C01832=1236.003,114.402,-48.327,-178.206,5.493,148.420
C01833=1235.998,114.651,-48.346,-178.204,5.494,148.419
C01834=1235.993,114.900,-48.366,-178.202,5.495,148.419
C01835=1235.989,115.150,-48.386,-178.199,5.496,148.418
C01836=1235.983,115.399,-48.405,-178.196,5.497,148.418
C01837=1235.979,115.648,-48.424,-178.194,5.498,148.417
C01838=1235.975,115.897,-48.444,-178.191,5.499,148.416
C01839=1235.969,116.146,-48.464,-178.189,5.500,148.416
C01840=1235.965,116.395,-48.483,-178.186,5.500,148.415
C01841=1235.960,116.645,-48.503,-178.183,5.502,148.415
C01842=1235.955,116.894,-48.522,-178.181,5.503,148.414
C01843=1235.950,117.143,-48.543,-178.178,5.503,148.414
C01844=1235.945,117.392,-48.562,-178.176,5.504,148.413
C01845=1235.940,117.641,-48.582,-178.174,5.505,148.413
C01846=1235.935,117.891,-48.601,-178.171,5.506,148.412
C01847=1235.932,118.139,-48.621,-178.168,5.507,148.412
C01848=1235.927,118.389,-48.641,-178.166,5.508,148.411
C01849=1235.921,118.638,-48.660,-178.163,5.509,148.410
C01850=1235.917,118.887,-48.680,-178.161,5.510,148.410
C01851=1235.912,119.136,-48.700,-178.158,5.511,148.409
C01852=1235.908,119.386,-48.720,-178.155,5.512,148.409
C01853=1235.903,119.634,-48.740,-178.153,5.513,148.408
C01854=1235.898,119.884,-48.759,-178.151,5.513,148.408
C01855=1235.893,120.133,-48.779,-178.148,5.514,148.407
C01856=1235.889,120.382,-48.799,-178.145,5.516,148.407
C01857=1235.883,120.631,-48.819,-178.143,5.517,148.406
C01858=1235.879,120.880,-48.838,-178.141,5.517,148.406
C01859=1235.874,121.129,-48.859,-178.138,5.518,148.405
C01860=1235.869,121.379,-48.878,-178.135,5.519,148.404
C01861=1235.864,121.627,-48.898,-178.133,5.521,148.404
C01862=1235.860,121.877,-48.918,-178.130,5.521,148.403
C01863=1235.855,122.126,-48.938,-178.128,5.522,148.403
C01864=1235.850,122.375,-48.958,-178.125,5.523,148.402
C01865=1235.845,122.624,-48.977,-178.122,5.524,148.402
C01866=1235.841,122.873,-48.998,-178.120,5.525,148.401
C01867=1235.836,123.123,-49.017,-178.117,5.526,148.401
C01868=1235.831,123.372,-49.038,-178.115,5.527,148.400
C01869=1235.827,123.621,-49.057,-178.113,5.528,148.399
C01870=1235.821,123.870,-49.078,-178.110,5.529,148.399
C01871=1235.816,124.119,-49.098,-178.107,5.530,148.398
C01872=1235.812,124.368,-49.118,-178.105,5.531,148.398
C01873=1235.807,124.618,-49.138,-178.102,5.531,148.397
C01874=1235.803,124.867,-49.158,-178.100,5.533,148.397
C01875=1235.798,125.116,-49.178,-178.097,5.534,148.396
C01876=1235.793,125.365,-49.198,-178.095,5.535,148.396
C01877=1235.788,125.614,-49.217,-178.092,5.535,148.395
C01878=1235.784,125.863,-49.238,-178.089,5.537,148.394
C01879=1235.779,126.113,-49.257,-178.087,5.538,148.394
C01880=1235.774,126.362,-49.278,-178.084,5.538,148.393
C01881=1235.769,126.611,-49.299,-178.082,5.539,148.393
C01882=1235.764,126.861,-49.318,-178.079,5.541,148.392
C01883=1235.759,127.109,-49.338,-178.076,5.542,148.392
C01884=1235.755,127.358,-49.358,-178.074,5.543,148.391
C01885=1235.750,127.607,-49.378,-178.072,5.543,148.391
C01886=1235.745,127.857,-49.399,-178.070,5.544,148.390
C01887=1235.740,128.106,-49.419,-178.066,5.546,148.390
C01888=1235.736,128.355,-49.439,-178.064,5.546,148.389
C01889=1235.731,128.604,-49.460,-178.062,5.547,148.389
C01890=1235.727,128.854,-49.480,-178.059,5.549,148.388
C01891=1235.722,129.102,-49.500,-178.056,5.550,148.388
C01892=1235.717,129.351,-49.520,-178.054,5.550,148.387
C01893=1235.712,129.601,-49.540,-178.052,5.551,148.387
C01894=1235.707,129.850,-49.561,-178.049,5.553,148.386
C01895=1235.703,130.099,-49.581,-178.046,5.553,148.385
C01896=1235.697,130.348,-49.601,-178.044,5.554,148.385
C01897=1235.693,130.597,-49.622,-178.041,5.555,148.384
C01898=1235.689,130.846,-49.642,-178.039,5.557,148.384
C01899=1235.684,131.095,-49.662,-178.036,5.558,148.383
C01900=1235.679,131.345,-49.683,-178.034,5.559,148.383
C01901=1235.674,131.594,-49.703,-178.031,5.559,148.382
C01902=1235.670,131.843,-49.723,-178.028,5.561,148.382
C01903=1235.665,132.091,-49.743,-178.026,5.562,148.381
C01904=1235.660,132.341,-49.764,-178.023,5.562,148.381
C01905=1235.655,132.590,-49.784,-178.021,5.564,148.380
C01906=1235.650,132.839,-49.804,-178.018,5.565,148.380
C01907=1235.645,133.088,-49.825,-178.016,5.566,148.379
C01908=1235.641,133.337,-49.846,-178.013,5.566,148.379
C01909=1235.635,133.606,-49.867,-178.010,5.568,148.378
C01910=1235.631,133.875,-49.889,-178.008,5.569,148.377
C01911=1235.626,134.143,-49.912,-178.005,5.570,148.377
C01912=1235.620,134.412,-49.934,-178.002,5.571,148.376
C01913=1235.616,134.661,-49.954,-177.999,5.572,148.376
C01914=1235.610,134.910,-49.975,-177.997,5.573,148.375
C01915=1235.606,135.159,-49.995,-177.995,5.574,148.375
C01916=1235.602,135.408,-50.016,-177.992,5.575,148.374
C01917=1235.596,135.658,-50.037,-177.989,5.577,148.374
C01918=1235.592,135.907,-50.057,-177.987,5.578,148.373
C01919=1235.588,136.156,-50.077,-177.985,5.578,148.373
C01920=1235.582,136.405,-50.098,-177.982,5.580,148.372
C01921=1235.578,136.654,-50.119,-177.979,5.581,148.372
C01922=1235.573,136.903,-50.140,-177.977,5.582,148.371
C01923=1235.568,137.152,-50.160,-177.974,5.583,148.371
C01924=1235.564,137.401,-50.180,-177.971,5.584,148.370
C01925=1235.559,137.650,-50.201,-177.969,5.585,148.370
C01926=1235.554,137.899,-50.222,-177.967,5.585,148.369
C01927=1235.549,138.148,-50.243,-177.964,5.587,148.369
C01928=1235.545,138.397,-50.263,-177.961,5.588,148.368
C01929=1235.539,138.647,-50.284,-177.959,5.589,148.368
C01930=1235.536,138.896,-50.305,-177.956,5.590,148.367
C01931=1235.530,139.145,-50.326,-177.954,5.591,148.367
C01932=1235.526,139.394,-50.346,-177.951,5.592,148.366
C01933=1235.521,139.644,-50.367,-177.949,5.594,148.366
C01934=1235.516,139.893,-50.387,-177.946,5.594,148.365
C01935=1235.512,140.142,-50.408,-177.944,5.595,148.364
C01936=1235.507,140.391,-50.429,-177.941,5.597,148.364
C01937=1235.502,140.640,-50.449,-177.939,5.598,148.363
C01938=1235.497,140.889,-50.470,-177.936,5.599,148.363
C01939=1235.493,141.138,-50.490,-177.934,5.600,148.362
C01940=1235.488,141.387,-50.512,-177.931,5.601,148.362
C01941=1235.483,141.636,-50.533,-177.929,5.602,148.361
C01942=1235.478,141.885,-50.553,-177.926,5.604,148.361
C01943=1235.474,142.135,-50.575,-177.923,5.604,148.360
C01944=1235.469,142.384,-50.595,-177.921,5.605,148.360
C01945=1235.464,142.633,-50.616,-177.918,5.607,148.359
C01946=1235.460,142.881,-50.637,-177.916,5.608,148.359
C01947=1235.455,143.131,-50.658,-177.913,5.608,148.358
C01948=1235.450,143.380,-50.679,-177.910,5.610,148.358
C01949=1235.445,143.629,-50.700,-177.908,5.611,148.357
C01950=1235.441,143.878,-50.720,-177.906,5.612,148.357
C01951=1235.436,144.127,-50.742,-177.903,5.613,148.356
C01952=1235.431,144.376,-50.763,-177.901,5.614,148.356
C01953=1235.427,144.625,-50.783,-177.898,5.615,148.355
C01954=1235.422,144.875,-50.804,-177.895,5.617,148.355
C01955=1235.418,145.123,-50.825,-177.893,5.617,148.354
C01956=1235.412,145.372,-50.846,-177.891,5.618,148.354
C01957=1235.407,145.621,-50.867,-177.887,5.620,148.353
C01958=1235.404,145.870,-50.889,-177.885,5.621,148.353
C01959=1235.399,146.120,-50.910,-177.883,5.622,148.352
C01960=1235.393,146.369,-50.931,-177.880,5.623,148.352
C01961=1235.389,146.617,-50.952,-177.878,5.624,148.351
C01962=1235.384,146.867,-50.973,-177.875,5.625,148.351
C01963=1235.379,147.116,-50.994,-177.873,5.627,148.350
C01964=1235.375,147.365,-51.015,-177.870,5.628,148.350
C01965=1235.370,147.614,-51.036,-177.867,5.629,148.349
C01966=1235.365,147.863,-51.057,-177.865,5.630,148.349
C01967=1235.361,148.112,-51.078,-177.863,5.631,148.348
C01968=1235.356,148.361,-51.099,-177.860,5.632,148.348
C01969=1235.351,148.610,-51.121,-177.857,5.633,148.347
C01970=1235.347,148.859,-51.142,-177.855,5.634,148.347
C01971=1235.342,149.109,-51.163,-177.852,5.636,148.346
C01972=1235.337,149.357,-51.184,-177.850,5.637,148.346
C01973=1235.332,149.607,-51.206,-177.847,5.638,148.345
C01974=1235.328,149.855,-51.227,-177.844,5.639,148.345
C01975=1235.323,150.105,-51.248,-177.842,5.640,148.344
C01976=1235.318,150.353,-51.269,-177.839,5.642,148.344
C01977=1235.313,150.603,-51.290,-177.837,5.643,148.343
C01978=1235.309,150.852,-51.312,-177.834,5.643,148.343
C01979=1235.304,151.101,-51.333,-177.832,5.645,148.342
C01980=1235.299,151.350,-51.354,-177.830,5.646,148.342
C01981=1235.294,151.599,-51.375,-177.826,5.648,148.341
C01982=1235.291,151.848,-51.397,-177.824,5.649,148.341
C01983=1235.286,152.097,-51.418,-177.822,5.649,148.340
C01984=1235.281,152.346,-51.439,-177.819,5.651,148.340
C01985=1235.276,152.596,-51.461,-177.817,5.652,148.339
C01986=1235.271,152.844,-51.482,-177.814,5.654,148.339
C01987=1235.266,153.093,-51.504,-177.811,5.654,148.338
C01988=1235.262,153.342,-51.524,-177.809,5.655,148.338
C01989=1235.258,153.591,-51.547,-177.806,5.657,148.337
C01990=1235.252,153.841,-51.568,-177.804,5.658,148.337
C01991=1235.248,154.089,-51.589,-177.801,5.660,148.337
C01992=1235.243,154.339,-51.611,-177.799,5.660,148.336
C01993=1235.238,154.588,-51.632,-177.797,5.661,148.336
C01994=1235.234,154.836,-51.653,-177.793,5.663,148.335
C01995=1235.229,155.085,-51.675,-177.791,5.664,148.335
C01996=1235.225,155.335,-51.696,-177.788,5.665,148.334
C01997=1235.220,155.583,-51.718,-177.786,5.666,148.334
C01998=1235.215,155.832,-51.740,-177.784,5.667,148.333
C01999=1235.210,156.082,-51.761,-177.781,5.669,148.333
C02000=1235.205,156.331,-51.783,-177.779,5.670,148.332
C02001=1235.201,156.579,-51.804,-177.776,5.671,148.332
C02002=1235.196,156.829,-51.826,-177.773,5.672,148.331
C02003=1235.191,157.078,-51.847,-177.770,5.674,148.331
C02004=1235.186,157.326,-51.869,-177.768,5.675,148.330
C02005=1235.183,157.575,-51.891,-177.766,5.676,148.330
C02006=1235.178,157.825,-51.911,-177.763,5.677,148.329
C02007=1235.173,158.073,-51.933,-177.761,5.678,148.329
C02008=1235.168,158.323,-51.955,-177.758,5.680,148.328
C02009=1235.164,158.571,-51.977,-177.756,5.681,148.328
C02010=1235.159,158.821,-51.999,-177.752,5.682,148.327
C02011=1235.154,159.070,-52.020,-177.750,5.683,148.327
C02012=1235.149,159.319,-52.042,-177.748,5.684,148.326
C02013=1235.144,159.587,-52.066,-177.745,5.686,148.326
C02014=1235.139,159.857,-52.089,-177.742,5.687,148.325
C02015=1235.134,160.126,-52.112,-177.740,5.688,148.325
C02016=1235.129,160.395,-52.136,-177.737,5.690,148.324
C02017=1235.124,160.644,-52.158,-177.735,5.691,148.324
C02018=1235.120,160.893,-52.180,-177.731,5.692,148.323
C02019=1235.115,161.142,-52.201,-177.729,5.693,148.323
C02020=1235.110,161.391,-52.223,-177.727,5.695,148.323
C02021=1235.106,161.640,-52.245,-177.724,5.696,148.322
C02022=1235.101,161.889,-52.266,-177.722,5.698,148.322
C02023=1235.097,162.138,-52.288,-177.719,5.698,148.321
C02024=1235.092,162.387,-52.310,-177.716,5.700,148.321
C02025=1235.087,162.636,-52.332,-177.714,5.701,148.320
C02026=1235.083,162.885,-52.354,-177.712,5.702,148.320
C02027=1235.078,163.134,-52.375,-177.709,5.704,148.319
C02028=1235.073,163.383,-52.398,-177.706,5.704,148.319
C02029=1235.068,163.632,-52.420,-177.704,5.706,148.318
C02030=1235.064,163.881,-52.442,-177.702,5.707,148.318
C02031=1235.059,164.130,-52.464,-177.698,5.709,148.317
C02032=1235.054,164.379,-52.486,-177.696,5.710,148.317
C02033=1235.050,164.628,-52.507,-177.693,5.711,148.316
C02034=1235.045,164.877,-52.529,-177.691,5.712,148.316
C02035=1235.040,165.126,-52.551,-177.688,5.714,148.316
C02036=1235.036,165.375,-52.573,-177.686,5.715,148.315
C02037=1235.031,165.624,-52.595,-177.683,5.716,148.315
C02038=1235.026,165.874,-52.617,-177.681,5.717,148.314
C02039=1235.021,166.122,-52.639,-177.678,5.719,148.314
C02040=1235.017,166.372,-52.661,-177.676,5.720,148.313
C02041=1235.012,166.620,-52.683,-177.673,5.721,148.313
C02042=1235.008,166.869,-52.706,-177.671,5.723,148.312
C02043=1235.003,167.118,-52.728,-177.669,5.724,148.312
C02044=1234.998,167.367,-52.750,-177.665,5.725,148.311
C02045=1234.994,167.616,-52.772,-177.663,5.726,148.311
C02046=1234.989,167.865,-52.794,-177.661,5.728,148.310
C02047=1234.984,168.114,-52.815,-177.658,5.729,148.310
C02048=1234.980,168.363,-52.839,-177.655,5.730,148.309
C02049=1234.975,168.611,-52.860,-177.653,5.731,148.309
C02050=1234.971,168.861,-52.882,-177.650,5.733,148.309
C02051=1234.966,169.109,-52.904,-177.648,5.734,148.308
C02052=1234.961,169.359,-52.927,-177.645,5.735,148.308
C02053=1234.957,169.608,-52.949,-177.643,5.736,148.307
C02054=1234.952,169.856,-52.971,-177.640,5.738,148.307
C02055=1234.948,170.106,-52.993,-177.638,5.739,148.306
C02056=1234.942,170.355,-53.015,-177.635,5.741,148.306
C02057=1234.938,170.604,-53.038,-177.633,5.742,148.305
C02058=1234.933,170.852,-53.060,-177.630,5.743,148.305
C02059=1234.928,171.102,-53.083,-177.628,5.744,148.304
C02060=1234.923,171.350,-53.104,-177.625,5.746,148.304
C02061=1234.919,171.599,-53.127,-177.622,5.747,148.303
C02062=1234.915,171.848,-53.149,-177.620,5.749,148.303
C02063=1234.910,172.097,-53.171,-177.618,5.750,148.303
C02064=1234.906,172.346,-53.194,-177.615,5.751,148.302
C02065=1234.901,172.595,-53.216,-177.612,5.752,148.302
C02066=1234.896,172.844,-53.238,-177.610,5.754,148.301
C02067=1234.892,173.093,-53.261,-177.607,5.755,148.301
C02068=1234.886,173.342,-53.283,-177.605,5.757,148.300
C02069=1234.882,173.591,-53.306,-177.602,5.758,148.300
C02070=1234.878,173.840,-53.328,-177.599,5.759,148.299
C02071=1234.872,174.089,-53.351,-177.597,5.761,148.299
C02072=1234.868,174.338,-53.373,-177.595,5.762,148.299
C02073=1234.863,174.586,-53.395,-177.591,5.763,148.298
C02074=1234.858,174.836,-53.418,-177.589,5.764,148.298
C02075=1234.854,175.085,-53.440,-177.587,5.766,148.297
C02076=1234.849,175.334,-53.463,-177.584,5.767,148.297
C02077=1234.845,175.583,-53.485,-177.581,5.769,148.296
C02078=1234.841,175.832,-53.508,-177.579,5.770,148.296
C02079=1234.835,176.080,-53.531,-177.576,5.771,148.295
C02080=1234.831,176.330,-53.553,-177.574,5.772,148.295
C02081=1234.826,176.579,-53.576,-177.571,5.774,148.295
C02082=1234.822,176.827,-53.598,-177.569,5.775,148.294
C02083=1234.817,177.076,-53.621,-177.566,5.777,148.294
C02084=1234.813,177.326,-53.643,-177.564,5.779,148.293
C02085=1234.807,177.574,-53.666,-177.562,5.780,148.293
C02086=1234.803,177.823,-53.688,-177.558,5.781,148.292
C02087=1234.798,178.072,-53.711,-177.556,5.782,148.292
C02088=1234.793,178.321,-53.733,-177.554,5.784,148.292
C02089=1234.789,178.570,-53.756,-177.551,5.785,148.291
C02090=1234.785,178.819,-53.779,-177.548,5.787,148.291
C02091=1234.780,179.068,-53.802,-177.546,5.788,148.290
C02092=1234.775,179.316,-53.824,-177.543,5.789,148.290
C02093=1234.770,179.566,-53.847,-177.541,5.791,148.289
C02094=1234.766,179.815,-53.870,-177.538,5.792,148.289
C02095=1234.761,180.063,-53.893,-177.536,5.794,148.289
C02096=1234.757,180.312,-53.915,-177.533,5.794,148.288
C02097=1234.752,180.561,-53.938,-177.531,5.796,148.288
C02098=1234.748,180.810,-53.961,-177.529,5.797,148.287
C02099=1234.742,181.059,-53.983,-177.525,5.799,148.287
C02100=1234.738,181.308,-54.006,-177.523,5.801,148.286
C02101=1234.734,181.557,-54.029,-177.521,5.802,148.286
C02102=1234.729,181.807,-54.052,-177.518,5.804,148.286
C02103=1234.724,182.055,-54.074,-177.515,5.804,148.285
C02104=1234.719,182.304,-54.098,-177.513,5.806,148.285
C02105=1234.715,182.552,-54.120,-177.511,5.807,148.284
C02106=1234.710,182.802,-54.143,-177.508,5.809,148.284
C02107=1234.706,183.051,-54.166,-177.505,5.810,148.283
C02108=1234.701,183.299,-54.189,-177.503,5.811,148.283
C02109=1234.696,183.548,-54.212,-177.500,5.813,148.283
C02110=1234.692,183.797,-54.234,-177.498,5.814,148.282
C02111=1234.688,184.046,-54.258,-177.495,5.816,148.282
C02112=1234.683,184.295,-54.281,-177.492,5.818,148.281
C02113=1234.678,184.543,-54.303,-177.490,5.819,148.281
C02114=1234.674,184.792,-54.327,-177.487,5.820,148.280
C02115=1234.669,185.042,-54.350,-177.485,5.821,148.280
C02116=1234.665,185.291,-54.372,-177.482,5.823,148.280
C02117=1234.659,185.561,-54.397,-177.479,5.825,148.279
C02118=1234.654,185.830,-54.423,-177.477,5.826,148.279
C02119=1234.650,186.099,-54.447,-177.474,5.827,148.278
C02120=1234.644,186.369,-54.472,-177.471,5.829,148.278
C02121=1234.640,186.618,-54.496,-177.469,5.831,148.277
C02122=1234.635,186.867,-54.519,-177.466,5.832,148.277
C02123=1234.631,187.116,-54.542,-177.464,5.833,148.277
C02124=1234.625,187.365,-54.564,-177.461,5.835,148.276
C02125=1234.621,187.614,-54.587,-177.459,5.836,148.276
C02126=1234.617,187.862,-54.610,-177.456,5.838,148.275
C02127=1234.612,188.112,-54.634,-177.454,5.839,148.275
C02128=1234.607,188.361,-54.657,-177.451,5.841,148.274
C02129=1234.603,188.610,-54.680,-177.448,5.843,148.274
C02130=1234.598,188.859,-54.704,-177.446,5.843,148.274
C02131=1234.594,189.107,-54.726,-177.443,5.845,148.273
C02132=1234.589,189.356,-54.749,-177.440,5.847,148.273
C02133=1234.584,189.605,-54.773,-177.438,5.848,148.272
C02134=1234.579,189.854,-54.796,-177.436,5.850,148.272
C02135=1234.575,190.103,-54.819,-177.433,5.850,148.272
C02136=1234.571,190.351,-54.842,-177.431,5.852,148.271
C02137=1234.566,190.601,-54.866,-177.428,5.854,148.271
C02138=1234.562,190.849,-54.890,-177.426,5.855,148.270
C02139=1234.557,191.098,-54.913,-177.423,5.857,148.270
C02140=1234.552,191.347,-54.936,-177.420,5.859,148.270
C02141=1234.547,191.596,-54.960,-177.418,5.860,148.269
C02142=1234.543,191.845,-54.983,-177.415,5.861,148.269
C02143=1234.538,192.093,-55.006,-177.413,5.862,148.268
C02144=1234.533,192.342,-55.029,-177.410,5.864,148.268
C02145=1234.529,192.591,-55.052,-177.407,5.866,148.268
C02146=1234.524,192.840,-55.076,-177.405,5.867,148.267
C02147=1234.520,193.089,-55.100,-177.403,5.869,148.267
C02148=1234.515,193.338,-55.123,-177.400,5.870,148.266
C02149=1234.510,193.587,-55.146,-177.398,5.871,148.266
C02150=1234.506,193.836,-55.170,-177.395,5.873,148.265
C02151=1234.502,194.084,-55.193,-177.392,5.875,148.265
C02152=1234.497,194.333,-55.217,-177.390,5.876,148.265
C02153=1234.493,194.582,-55.240,-177.387,5.878,148.264
C02154=1234.488,194.831,-55.263,-177.384,5.879,148.264
C02155=1234.483,195.080,-55.287,-177.382,5.880,148.263
C02156=1234.479,195.328,-55.311,-177.380,5.882,148.263
C02157=1234.474,195.577,-55.334,-177.377,5.884,148.263
C02158=1234.469,195.826,-55.357,-177.374,5.885,148.262
C02159=1234.465,196.075,-55.381,-177.372,5.887,148.262
C02160=1234.460,196.324,-55.405,-177.369,5.889,148.262
C02161=1234.456,196.573,-55.428,-177.367,5.890,148.261
C02162=1234.451,196.822,-55.452,-177.364,5.891,148.261
C02163=1234.446,197.070,-55.476,-177.361,5.893,148.260
C02164=1234.442,197.319,-55.499,-177.359,5.894,148.260
C02165=1234.437,197.568,-55.522,-177.357,5.896,148.260
C02166=1234.433,197.817,-55.546,-177.354,5.898,148.259
C02167=1234.428,198.066,-55.570,-177.352,5.899,148.259
C02168=1234.423,198.315,-55.593,-177.349,5.900,148.258
C02169=1234.419,198.563,-55.617,-177.346,5.902,148.258
C02170=1234.414,198.812,-55.641,-177.344,5.903,148.258
C02171=1234.410,199.061,-55.665,-177.341,5.905,148.257
C02172=1234.405,199.310,-55.688,-177.339,5.907,148.257
C02173=1234.400,199.559,-55.711,-177.337,5.908,148.256
C02174=1234.396,199.807,-55.735,-177.334,5.909,148.256
C02175=1234.391,200.057,-55.759,-177.331,5.911,148.256
C02176=1234.387,200.306,-55.784,-177.328,5.913,148.255
C02177=1234.382,200.555,-55.807,-177.326,5.914,148.255
C02178=1234.378,200.803,-55.831,-177.324,5.916,148.255
C02179=1234.373,201.052,-55.855,-177.321,5.918,148.254
C02180=1234.369,201.301,-55.879,-177.318,5.919,148.254
C02181=1234.364,201.550,-55.902,-177.316,5.920,148.253
C02182=1234.359,201.798,-55.926,-177.313,5.922,148.253
C02183=1234.355,202.047,-55.950,-177.311,5.923,148.253
C02184=1234.350,202.296,-55.974,-177.308,5.925,148.252
C02185=1234.345,202.545,-55.998,-177.306,5.927,148.252
C02186=1234.341,202.794,-56.022,-177.303,5.929,148.251
C02187=1234.337,203.042,-56.046,-177.301,5.930,148.251
C02188=1234.332,203.291,-56.069,-177.298,5.932,148.251
C02189=1234.328,203.540,-56.094,-177.295,5.933,148.250
C02190=1234.322,203.789,-56.117,-177.293,5.934,148.250
C02191=1234.318,204.037,-56.142,-177.291,5.936,148.250
C02192=1234.313,204.286,-56.166,-177.288,5.938,148.249
C02193=1234.309,204.535,-56.189,-177.285,5.940,148.249
C02194=1234.305,204.784,-56.213,-177.283,5.941,148.248
C02195=1234.300,205.033,-56.238,-177.280,5.943,148.248
C02196=1234.295,205.282,-56.261,-177.278,5.944,148.248
C02197=1234.291,205.530,-56.286,-177.275,5.945,148.247
C02198=1234.286,205.779,-56.310,-177.273,5.947,148.247
C02199=1234.281,206.028,-56.334,-177.270,5.949,148.247
C02200=1234.277,206.277,-56.358,-177.267,5.951,148.246
C02201=1234.273,206.526,-56.382,-177.265,5.952,148.246
C02202=1234.268,206.775,-56.405,-177.262,5.954,148.245
C02203=1234.263,207.023,-56.430,-177.260,5.955,148.245
C02204=1234.258,207.272,-56.454,-177.257,5.957,148.245
C02205=1234.255,207.521,-56.479,-177.255,5.958,148.244
C02206=1234.249,207.770,-56.503,-177.252,5.960,148.244
C02207=1234.245,208.019,-56.527,-177.250,5.962,148.244
C02208=1234.240,208.267,-56.551,-177.247,5.964,148.243
C02209=1234.236,208.515,-56.575,-177.245,5.965,148.243
C02210=1234.231,208.765,-56.600,-177.242,5.967,148.242
C02211=1234.227,209.014,-56.623,-177.239,5.968,148.242
C02212=1234.222,209.262,-56.647,-177.237,5.970,148.242
C02213=1234.217,209.511,-56.672,-177.235,5.971,148.241
C02214=1234.213,209.760,-56.696,-177.232,5.973,148.241
C02215=1234.208,210.009,-56.721,-177.229,5.975,148.241
C02216=1234.204,210.257,-56.745,-177.226,5.977,148.240
C02217=1234.200,210.506,-56.769,-177.224,5.978,148.240
C02218=1234.194,210.755,-56.793,-177.222,5.979,148.239
C02219=1234.190,211.004,-56.818,-177.219,5.981,148.239
C02220=1234.186,211.252,-56.842,-177.216,5.983,148.239
C02221=1234.181,211.523,-56.868,-177.214,5.985,148.238
C02222=1234.176,211.793,-56.895,-177.211,5.987,148.238
C02223=1234.171,212.064,-56.922,-177.208,5.988,148.237
C02224=1234.166,212.334,-56.948,-177.205,5.990,148.237
C02225=1234.161,212.583,-56.972,-177.203,5.992,148.237
C02226=1234.156,212.832,-56.997,-177.201,5.993,148.236
C02227=1234.152,213.081,-57.021,-177.198,5.995,148.236
C02228=1234.147,213.329,-57.046,-177.195,5.997,148.236
C02229=1234.143,213.578,-57.070,-177.192,5.999,148.235
C02230=1234.139,213.827,-57.095,-177.190,6.000,148.235
C02231=1234.134,214.076,-57.119,-177.188,6.001,148.234
C02232=1234.129,214.324,-57.143,-177.185,6.003,148.234
C02233=1234.125,214.574,-57.168,-177.182,6.005,148.234
C02234=1234.121,214.822,-57.192,-177.180,6.007,148.234
C02235=1234.116,215.070,-57.218,-177.178,6.008,148.233
C02236=1234.112,215.319,-57.242,-177.175,6.010,148.233
C02237=1234.107,215.568,-57.267,-177.172,6.012,148.232
C02238=1234.102,215.816,-57.291,-177.170,6.014,148.232
C02239=1234.098,216.066,-57.316,-177.167,6.016,148.232
C02240=1234.093,216.314,-57.341,-177.164,6.016,148.231
C02241=1234.088,216.563,-57.365,-177.162,6.018,148.231
C02242=1234.084,216.812,-57.390,-177.159,6.020,148.231
C02243=1234.080,217.060,-57.415,-177.157,6.022,148.230
C02244=1234.075,217.309,-57.439,-177.154,6.024,148.230
C02245=1234.071,217.558,-57.464,-177.152,6.025,148.230
C02246=1234.066,217.807,-57.488,-177.149,6.027,148.229
C02247=1234.062,218.056,-57.513,-177.147,6.029,148.229
C02248=1234.057,218.304,-57.538,-177.144,6.030,148.229
C02249=1234.052,218.553,-57.563,-177.141,6.032,148.228
C02250=1234.048,218.802,-57.587,-177.139,6.033,148.228
C02251=1234.043,219.050,-57.612,-177.137,6.035,148.228
C02252=1234.038,219.300,-57.637,-177.134,6.037,148.227
C02253=1234.034,219.548,-57.662,-177.131,6.039,148.227
C02254=1234.029,219.796,-57.686,-177.129,6.041,148.227
C02255=1234.025,220.045,-57.711,-177.127,6.042,148.226
C02256=1234.021,220.294,-57.736,-177.124,6.044,148.226
C02257=1234.016,220.543,-57.761,-177.122,6.046,148.226
C02258=1234.012,220.791,-57.785,-177.118,6.047,148.225
C02259=1234.007,221.040,-57.811,-177.116,6.049,148.225
C02260=1234.002,221.289,-57.836,-177.113,6.051,148.224
C02261=1233.998,221.537,-57.860,-177.111,6.052,148.224
C02262=1233.994,221.786,-57.886,-177.109,6.054,148.224
C02263=1233.989,222.035,-57.910,-177.106,6.056,148.223
C02264=1233.984,222.284,-57.935,-177.103,6.058,148.223
C02265=1233.980,222.532,-57.960,-177.101,6.059,148.223
C02266=1233.975,222.782,-57.985,-177.099,6.060,148.222
C02267=1233.971,223.030,-58.011,-177.096,6.062,148.222
C02268=1233.967,223.279,-58.035,-177.093,6.064,148.222
C02269=1233.962,223.527,-58.060,-177.091,6.066,148.221
C02270=1233.957,223.776,-58.085,-177.088,6.068,148.221
C02271=1233.952,224.025,-58.110,-177.085,6.070,148.221
C02272=1233.949,224.274,-58.135,-177.083,6.071,148.220
C02273=1233.944,224.522,-58.160,-177.081,6.073,148.220
C02274=1233.939,224.771,-58.186,-177.078,6.075,148.220
C02275=1233.934,225.020,-58.210,-177.076,6.076,148.219
C02276=1233.930,225.269,-58.236,-177.073,6.078,148.219
C02277=1233.926,225.517,-58.260,-177.070,6.080,148.219
C02278=1233.922,225.766,-58.286,-177.068,6.081,148.218
C02279=1233.916,226.015,-58.311,-177.066,6.083,148.218
C02280=1233.912,226.263,-58.336,-177.063,6.085,148.218
C02281=1233.907,226.511,-58.362,-177.060,6.087,148.217
C02282=1233.904,226.761,-58.386,-177.058,6.089,148.217
C02283=1233.899,227.009,-58.411,-177.055,6.091,148.217
C02284=1233.894,227.258,-58.437,-177.053,6.092,148.216
C02285=1233.889,227.506,-58.462,-177.050,6.094,148.216
C02286=1233.885,227.755,-58.488,-177.048,6.095,148.216
C02287=1233.880,228.004,-58.512,-177.045,6.097,148.215
C02288=1233.876,228.252,-58.538,-177.043,6.099,148.215
C02289=1233.871,228.501,-58.563,-177.040,6.101,148.215
C02290=1233.867,228.750,-58.588,-177.037,6.103,148.214
C02291=1233.863,228.999,-58.614,-177.035,6.104,148.214
C02292=1233.858,229.247,-58.638,-177.033,6.106,148.214
C02293=1233.854,229.496,-58.664,-177.030,6.108,148.213
C02294=1233.849,229.744,-58.689,-177.027,6.110,148.213
C02295=1233.845,229.993,-58.715,-177.025,6.112,148.213
C02296=1233.840,230.242,-58.740,-177.022,6.113,148.212
C02297=1233.835,230.490,-58.766,-177.020,6.116,148.212
C02298=1233.831,230.739,-58.791,-177.018,6.117,148.212
C02299=1233.826,230.987,-58.817,-177.015,6.118,148.212
C02300=1233.822,231.237,-58.842,-177.013,6.120,148.211
C02301=1233.817,231.486,-58.868,-177.010,6.122,148.211
C02302=1233.813,231.734,-58.893,-177.008,6.124,148.211
C02303=1233.808,231.983,-58.919,-177.005,6.126,148.210
C02304=1233.803,232.231,-58.944,-177.002,6.128,148.210
C02305=1233.799,232.480,-58.969,-177.000,6.129,148.210
C02306=1233.795,232.729,-58.995,-176.998,6.131,148.209
C02307=1233.790,232.977,-59.020,-176.995,6.133,148.209
C02308=1233.786,233.226,-59.046,-176.992,6.135,148.209
C02309=1233.781,233.475,-59.072,-176.990,6.136,148.208
C02310=1233.777,233.723,-59.097,-176.987,6.138,148.208
C02311=1233.772,233.972,-59.122,-176.985,6.140,148.208
C02312=1233.768,234.221,-59.148,-176.982,6.142,148.208
C02313=1233.763,234.469,-59.173,-176.980,6.143,148.207
C02314=1233.759,234.718,-59.199,-176.977,6.145,148.207
C02315=1233.755,234.967,-59.225,-176.975,6.147,148.207
C02316=1233.750,235.215,-59.250,-176.972,6.149,148.206
C02317=1233.746,235.464,-59.276,-176.970,6.151,148.206
C02318=1233.741,235.712,-59.302,-176.967,6.153,148.206
C02319=1233.736,235.960,-59.327,-176.965,6.155,148.205
C02320=1233.732,236.209,-59.353,-176.962,6.157,148.205
C02321=1233.727,236.458,-59.379,-176.960,6.158,148.205
C02322=1233.722,236.706,-59.405,-176.957,6.160,148.204
C02323=1233.718,236.955,-59.430,-176.955,6.161,148.204
C02324=1233.714,237.204,-59.456,-176.952,6.163,148.204
C02325=1233.709,237.475,-59.484,-176.949,6.165,148.204
C02326=1233.704,237.747,-59.512,-176.947,6.167,148.203
C02327=1233.700,238.018,-59.541,-176.944,6.170,148.203
C02328=1233.694,238.290,-59.568,-176.941,6.172,148.203
C02329=1233.690,238.538,-59.594,-176.939,6.174,148.202
C02330=1233.685,238.788,-59.620,-176.936,6.175,148.202
C02331=1233.681,239.035,-59.646,-176.934,6.177,148.202
C02332=1233.676,239.284,-59.672,-176.931,6.178,148.201
C02333=1233.672,239.533,-59.698,-176.929,6.181,148.201
C02334=1233.668,239.781,-59.724,-176.926,6.182,148.201
C02335=1233.662,240.030,-59.750,-176.924,6.184,148.201
C02336=1233.658,240.279,-59.775,-176.921,6.186,148.200
C02337=1233.654,240.527,-59.801,-176.919,6.188,148.200
C02338=1233.650,240.776,-59.828,-176.916,6.190,148.200
C02339=1233.646,241.024,-59.853,-176.913,6.192,148.199
C02340=1233.640,241.273,-59.879,-176.911,6.194,148.199
C02341=1233.636,241.522,-59.905,-176.909,6.196,148.199
C02342=1233.632,241.770,-59.931,-176.907,6.197,148.199
C02343=1233.628,242.019,-59.957,-176.904,6.199,148.198
C02344=1233.622,242.267,-59.983,-176.901,6.201,148.198
C02345=1233.618,242.516,-60.009,-176.899,6.203,148.198
C02346=1233.614,242.765,-60.035,-176.896,6.205,148.197
C02347=1233.609,243.013,-60.062,-176.894,6.206,148.197
C02348=1233.605,243.262,-60.088,-176.891,6.208,148.197
C02349=1233.601,243.511,-60.113,-176.889,6.211,148.197
C02350=1233.595,243.759,-60.139,-176.886,6.212,148.196
C02351=1233.591,244.007,-60.166,-176.884,6.214,148.196
C02352=1233.587,244.256,-60.192,-176.881,6.216,148.196
C02353=1233.582,244.505,-60.218,-176.878,6.218,148.195
C02354=1233.578,244.754,-60.244,-176.876,6.219,148.195
C02355=1233.574,245.002,-60.270,-176.874,6.221,148.195
C02356=1233.569,245.250,-60.297,-176.872,6.223,148.195
C02357=1233.564,245.499,-60.323,-176.869,6.225,148.194
C02358=1233.560,245.748,-60.348,-176.866,6.227,148.194
C02359=1233.556,245.996,-60.375,-176.864,6.229,148.194
C02360=1233.551,246.245,-60.401,-176.861,6.231,148.193
C02361=1233.547,246.494,-60.428,-176.859,6.233,148.193
C02362=1233.542,246.742,-60.454,-176.856,6.235,148.193
C02363=1233.538,246.991,-60.480,-176.854,6.237,148.193
C02364=1233.533,247.239,-60.506,-176.851,6.239,148.192
C02365=1233.529,247.488,-60.532,-176.849,6.241,148.192
C02366=1233.524,247.736,-60.559,-176.846,6.242,148.192
C02367=1233.520,247.985,-60.585,-176.844,6.245,148.192
C02368=1233.515,248.234,-60.612,-176.841,6.247,148.191
C02369=1233.511,248.482,-60.638,-176.839,6.248,148.191
C02370=1233.506,248.731,-60.665,-176.836,6.250,148.191
C02371=1233.502,248.980,-60.691,-176.834,6.251,148.190
C02372=1233.498,249.228,-60.717,-176.832,6.254,148.190
C02373=1233.494,249.476,-60.744,-176.829,6.255,148.190
C02374=1233.489,249.725,-60.770,-176.827,6.257,148.190
C02375=1233.485,249.974,-60.797,-176.824,6.259,148.189
C02376=1233.480,250.222,-60.822,-176.821,6.261,148.189
C02377=1233.475,250.470,-60.849,-176.819,6.263,148.189
C02378=1233.470,250.719,-60.876,-176.817,6.265,148.189
C02379=1233.466,250.967,-60.902,-176.814,6.267,148.188
C02380=1233.462,251.216,-60.929,-176.811,6.269,148.188
C02381=1233.457,251.465,-60.955,-176.809,6.271,148.188
C02382=1233.453,251.713,-60.982,-176.807,6.273,148.188
C02383=1233.449,251.961,-61.009,-176.804,6.275,148.187
C02384=1233.444,252.211,-61.035,-176.802,6.277,148.187
C02385=1233.440,252.459,-61.061,-176.799,6.279,148.187
C02386=1233.435,252.707,-61.088,-176.796,6.281,148.186
C02387=1233.430,252.956,-61.115,-176.794,6.283,148.186
C02388=1233.426,253.205,-61.141,-176.792,6.285,148.186
C02389=1233.422,253.453,-61.168,-176.789,6.287,148.186
C02390=1233.418,253.701,-61.195,-176.786,6.289,148.185
C02391=1233.413,253.950,-61.221,-176.784,6.291,148.185
C02392=1233.408,254.199,-61.248,-176.782,6.293,148.185
C02393=1233.404,254.447,-61.275,-176.779,6.295,148.185
C02394=1233.400,254.696,-61.302,-176.776,6.296,148.184
C02395=1233.396,254.944,-61.328,-176.774,6.299,148.184
C02396=1233.391,255.193,-61.354,-176.772,6.301,148.184
C02397=1233.386,255.441,-61.382,-176.769,6.302,148.184
C02398=1233.382,255.690,-61.408,-176.767,6.304,148.183
C02399=1233.378,255.938,-61.435,-176.764,6.307,148.183
C02400=1233.373,256.187,-61.462,-176.762,6.308,148.183
C02401=1233.369,256.435,-61.489,-176.759,6.310,148.183
C02402=1233.365,256.685,-61.515,-176.757,6.312,148.183
C02403=1233.360,256.933,-61.542,-176.754,6.314,148.182
C02404=1233.355,257.182,-61.569,-176.752,6.316,148.182
C02405=1233.351,257.430,-61.596,-176.749,6.318,148.182
C02406=1233.347,257.678,-61.623,-176.747,6.320,148.182
C02407=1233.342,257.927,-61.650,-176.745,6.322,148.181
C02408=1233.337,258.175,-61.677,-176.742,6.324,148.181
C02409=1233.333,258.423,-61.704,-176.739,6.326,148.181
C02410=1233.329,258.672,-61.731,-176.737,6.328,148.181
C02411=1233.324,258.920,-61.758,-176.735,6.330,148.180
C02412=1233.320,259.169,-61.785,-176.732,6.332,148.180
C02413=1233.316,259.417,-61.811,-176.729,6.334,148.180
C02414=1233.312,259.666,-61.839,-176.727,6.336,148.180
C02415=1233.307,259.915,-61.866,-176.725,6.338,148.179
C02416=1233.302,260.163,-61.893,-176.722,6.340,148.179
C02417=1233.298,260.411,-61.919,-176.720,6.342,148.179
C02418=1233.294,260.660,-61.946,-176.717,6.344,148.179
C02419=1233.289,260.908,-61.973,-176.715,6.346,148.178
C02420=1233.284,261.157,-62.000,-176.713,6.348,148.178
C02421=1233.280,261.405,-62.027,-176.710,6.350,148.178
C02422=1233.276,261.655,-62.055,-176.707,6.352,148.178
C02423=1233.272,261.903,-62.081,-176.705,6.354,148.178
C02424=1233.267,262.151,-62.108,-176.703,6.356,148.177
C02425=1233.262,262.400,-62.135,-176.700,6.358,148.177
C02426=1233.258,262.648,-62.163,-176.698,6.360,148.177
C02427=1233.253,262.896,-62.190,-176.695,6.362,148.177
C02428=1233.249,263.145,-62.218,-176.693,6.364,148.176
C02429=1233.245,263.418,-62.247,-176.690,6.366,148.176
C02430=1233.239,263.691,-62.277,-176.687,6.369,148.176
C02431=1233.235,263.963,-62.307,-176.685,6.371,148.176
C02432=1233.230,264.236,-62.336,-176.682,6.373,148.176
C02433=1233.226,264.484,-62.364,-176.680,6.375,148.175
C02434=1233.221,264.732,-62.391,-176.677,6.377,148.175
C02435=1233.217,264.980,-62.418,-176.674,6.380,148.175
C02436=1233.212,265.230,-62.446,-176.672,6.381,148.175
C02437=1233.208,265.478,-62.473,-176.669,6.383,148.174
C02438=1233.203,265.726,-62.501,-176.667,6.386,148.174
C02439=1233.199,265.974,-62.528,-176.665,6.387,148.174
C02440=1233.194,266.223,-62.555,-176.662,6.390,148.174
C02441=1233.190,266.472,-62.582,-176.660,6.392,148.174
C02442=1233.186,266.720,-62.610,-176.657,6.394,148.173
C02443=1233.181,266.968,-62.637,-176.655,6.396,148.173
C02444=1233.176,267.217,-62.664,-176.653,6.398,148.173
C02445=1233.173,267.466,-62.692,-176.650,6.400,148.173
C02446=1233.168,267.714,-62.719,-176.648,6.402,148.173
C02447=1233.163,267.963,-62.746,-176.645,6.404,148.172
C02448=1233.159,268.210,-62.774,-176.643,6.406,148.172
C02449=1233.155,268.460,-62.802,-176.641,6.408,148.172
C02450=1233.151,268.708,-62.829,-176.638,6.410,148.172
C02451=1233.146,268.956,-62.856,-176.636,6.412,148.171
C02452=1233.142,269.205,-62.884,-176.633,6.414,148.171
C02453=1233.138,269.453,-62.912,-176.630,6.416,148.171
C02454=1233.133,269.702,-62.939,-176.628,6.419,148.171
C02455=1233.129,269.949,-62.966,-176.625,6.421,148.171
C02456=1233.124,270.199,-62.994,-176.623,6.423,148.170
C02457=1233.119,270.447,-63.022,-176.621,6.425,148.170
C02458=1233.115,270.695,-63.049,-176.618,6.427,148.170
C02459=1233.111,270.944,-63.077,-176.616,6.429,148.170
C02460=1233.106,271.192,-63.105,-176.613,6.431,148.170
C02461=1233.102,271.440,-63.132,-176.611,6.433,148.169
C02462=1233.098,271.689,-63.160,-176.609,6.435,148.169
C02463=1233.094,271.937,-63.187,-176.606,6.437,148.169
C02464=1233.088,272.186,-63.215,-176.604,6.439,148.169
C02465=1233.084,272.435,-63.243,-176.601,6.441,148.169
C02466=1233.080,272.683,-63.271,-176.599,6.444,148.168
C02467=1233.075,272.931,-63.298,-176.596,6.446,148.168
C02468=1233.072,273.180,-63.326,-176.594,6.448,148.168
C02469=1233.067,273.428,-63.353,-176.591,6.450,148.168
C02470=1233.062,273.676,-63.382,-176.589,6.452,148.168
C02471=1233.058,273.925,-63.410,-176.587,6.454,148.167
C02472=1233.054,274.173,-63.437,-176.584,6.456,148.167
C02473=1233.049,274.421,-63.465,-176.582,6.458,148.167
C02474=1233.045,274.670,-63.493,-176.579,6.460,148.167
C02475=1233.040,274.919,-63.520,-176.577,6.462,148.167
C02476=1233.036,275.167,-63.548,-176.575,6.464,148.166
C02477=1233.032,275.415,-63.576,-176.572,6.467,148.166
C02478=1233.027,275.664,-63.603,-176.569,6.469,148.166
C02479=1233.023,275.913,-63.632,-176.567,6.471,148.166
C02480=1233.018,276.160,-63.660,-176.565,6.473,148.166
C02481=1233.014,276.408,-63.688,-176.563,6.475,148.166
C02482=1233.010,276.657,-63.715,-176.560,6.477,148.165
C02483=1233.005,276.906,-63.744,-176.558,6.480,148.165
C02484=1233.001,277.154,-63.772,-176.555,6.482,148.165
C02485=1232.997,277.402,-63.799,-176.553,6.484,148.165
C02486=1232.992,277.651,-63.828,-176.550,6.486,148.165
C02487=1232.988,277.899,-63.855,-176.548,6.489,148.165
C02488=1232.983,278.147,-63.883,-176.545,6.491,148.164
C02489=1232.979,278.396,-63.912,-176.543,6.493,148.164
C02490=1232.975,278.644,-63.940,-176.541,6.495,148.164
C02491=1232.971,278.893,-63.968,-176.538,6.497,148.164
C02492=1232.966,279.141,-63.996,-176.536,6.499,148.164
C02493=1232.962,279.390,-64.024,-176.534,6.501,148.164
C02494=1232.957,279.638,-64.051,-176.531,6.504,148.163
C02495=1232.953,279.887,-64.080,-176.529,6.506,148.163
C02496=1232.948,280.135,-64.108,-176.526,6.508,148.163
C02497=1232.945,280.383,-64.136,-176.524,6.510,148.163
C02498=1232.940,280.631,-64.164,-176.521,6.512,148.163
C02499=1232.936,280.880,-64.192,-176.519,6.514,148.163
C02500=1232.931,281.128,-64.221,-176.517,6.516,148.162
C02501=1232.927,281.377,-64.249,-176.514,6.518,148.162
C02502=1232.923,281.625,-64.277,-176.511,6.521,148.162
C02503=1232.918,281.874,-64.305,-176.509,6.523,148.162
C02504=1232.914,282.121,-64.333,-176.507,6.525,148.162
C02505=1232.909,282.370,-64.362,-176.504,6.527,148.162
C02506=1232.905,282.618,-64.390,-176.502,6.530,148.162
C02507=1232.900,282.867,-64.419,-176.500,6.532,148.161
C02508=1232.896,283.115,-64.446,-176.498,6.534,148.161
C02509=1232.892,283.364,-64.475,-176.495,6.537,148.161
C02510=1232.887,283.612,-64.503,-176.492,6.539,148.161
C02511=1232.883,283.861,-64.532,-176.490,6.541,148.161
C02512=1232.878,284.109,-64.559,-176.488,6.543,148.160
C02513=1232.874,284.357,-64.588,-176.486,6.545,148.160
C02514=1232.870,284.605,-64.617,-176.483,6.547,148.160
C02515=1232.865,284.854,-64.645,-176.481,6.549,148.160
C02516=1232.861,285.101,-64.673,-176.478,6.552,148.160
C02517=1232.857,285.350,-64.702,-176.476,6.554,148.160
C02518=1232.853,285.599,-64.730,-176.474,6.556,148.160
C02519=1232.848,285.847,-64.758,-176.471,6.558,148.159
C02520=1232.844,286.096,-64.786,-176.469,6.561,148.159
C02521=1232.839,286.343,-64.816,-176.466,6.562,148.159
C02522=1232.835,286.592,-64.844,-176.464,6.566,148.159
C02523=1232.830,286.840,-64.872,-176.462,6.568,148.159
C02524=1232.826,287.089,-64.901,-176.459,6.570,148.159
C02525=1232.822,287.337,-64.930,-176.457,6.572,148.159
C02526=1232.817,287.585,-64.958,-176.454,6.574,148.158
C02527=1232.814,287.834,-64.986,-176.452,6.576,148.158
C02528=1232.809,288.082,-65.015,-176.449,6.579,148.158
C02529=1232.804,288.330,-65.044,-176.447,6.581,148.158
C02530=1232.801,288.579,-65.072,-176.445,6.583,148.158
C02531=1232.796,288.827,-65.101,-176.443,6.585,148.158
C02532=1232.791,289.075,-65.130,-176.440,6.587,148.158
C02533=1232.787,289.349,-65.161,-176.437,6.590,148.158
C02534=1232.782,289.623,-65.192,-176.435,6.592,148.157
C02535=1232.777,289.897,-65.224,-176.432,6.595,148.157
C02536=1232.772,290.171,-65.256,-176.430,6.597,148.157
C02537=1232.768,290.420,-65.285,-176.427,6.599,148.157
C02538=1232.763,290.668,-65.313,-176.425,6.603,148.157
C02539=1232.759,290.917,-65.342,-176.422,6.604,148.157
C02540=1232.755,291.165,-65.371,-176.420,6.607,148.157
C02541=1232.750,291.413,-65.399,-176.418,6.609,148.157
C02542=1232.747,291.661,-65.428,-176.415,6.611,148.156
C02543=1232.742,291.910,-65.457,-176.413,6.613,148.156
C02544=1232.737,292.157,-65.486,-176.411,6.616,148.156
C02545=1232.733,292.406,-65.515,-176.408,6.618,148.156
C02546=1232.729,292.654,-65.544,-176.406,6.620,148.156
C02547=1232.724,292.902,-65.572,-176.404,6.622,148.156
C02548=1232.720,293.151,-65.601,-176.402,6.625,148.156
C02549=1232.716,293.400,-65.630,-176.399,6.627,148.155
C02550=1232.712,293.648,-65.659,-176.397,6.630,148.155
C02551=1232.707,293.896,-65.687,-176.394,6.632,148.155
C02552=1232.703,294.144,-65.717,-176.392,6.634,148.155
C02553=1232.698,294.393,-65.746,-176.390,6.636,148.155
C02554=1232.694,294.640,-65.775,-176.387,6.639,148.155
C02555=1232.690,294.889,-65.803,-176.385,6.641,148.155
C02556=1232.686,295.137,-65.832,-176.382,6.643,148.155
C02557=1232.681,295.386,-65.862,-176.380,6.645,148.155
C02558=1232.676,295.634,-65.890,-176.378,6.648,148.155
C02559=1232.672,295.882,-65.920,-176.376,6.651,148.155
C02560=1232.668,296.131,-65.948,-176.373,6.653,148.154
C02561=1232.664,296.379,-65.977,-176.371,6.655,148.154
C02562=1232.659,296.626,-66.006,-176.369,6.657,148.154
C02563=1232.655,296.875,-66.035,-176.367,6.659,148.154
C02564=1232.651,297.124,-66.064,-176.364,6.662,148.154
C02565=1232.647,297.372,-66.094,-176.361,6.664,148.154
C02566=1232.642,297.620,-66.123,-176.359,6.666,148.154
C02567=1232.637,297.868,-66.152,-176.357,6.669,148.154
C02568=1232.633,298.117,-66.181,-176.355,6.671,148.154
C02569=1232.630,298.365,-66.210,-176.352,6.674,148.153
C02570=1232.625,298.613,-66.239,-176.350,6.676,148.153
C02571=1232.621,298.862,-66.268,-176.348,6.678,148.153
C02572=1232.616,299.109,-66.297,-176.346,6.680,148.153
C02573=1232.612,299.357,-66.327,-176.344,6.683,148.153
C02574=1232.608,299.606,-66.356,-176.340,6.685,148.153
C02575=1232.603,299.855,-66.385,-176.338,6.688,148.153
C02576=1232.599,300.103,-66.414,-176.336,6.690,148.153
C02577=1232.594,300.350,-66.444,-176.334,6.692,148.153
C02578=1232.590,300.599,-66.473,-176.331,6.695,148.153
C02579=1232.586,300.847,-66.502,-176.329,6.697,148.153
C02580=1232.582,301.095,-66.532,-176.327,6.699,148.152
C02581=1232.577,301.344,-66.561,-176.325,6.701,148.152
C02582=1232.573,301.592,-66.590,-176.323,6.704,148.152
C02583=1232.569,301.841,-66.620,-176.320,6.707,148.152
C02584=1232.564,302.088,-66.649,-176.318,6.709,148.152
C02585=1232.560,302.337,-66.678,-176.316,6.711,148.152
C02586=1232.556,302.585,-66.708,-176.314,6.713,148.152
C02587=1232.552,302.833,-66.737,-176.310,6.716,148.152
C02588=1232.548,303.081,-66.766,-176.308,6.718,148.152
C02589=1232.543,303.330,-66.796,-176.306,6.721,148.152
C02590=1232.539,303.578,-66.825,-176.304,6.723,148.152
C02591=1232.534,303.825,-66.854,-176.302,6.725,148.152
C02592=1232.529,304.074,-66.884,-176.299,6.728,148.152
C02593=1232.525,304.322,-66.914,-176.297,6.730,148.152
C02594=1232.521,304.571,-66.943,-176.295,6.733,148.152
C02595=1232.517,304.819,-66.973,-176.293,6.735,148.152
C02596=1232.513,305.067,-67.002,-176.290,6.737,148.151
C02597=1232.509,305.315,-67.032,-176.288,6.740,148.151
C02598=1232.504,305.564,-67.061,-176.286,6.742,148.151
C02599=1232.500,305.812,-67.091,-176.284,6.744,148.151
C02600=1232.496,306.060,-67.120,-176.281,6.747,148.151
C02601=1232.491,306.309,-67.150,-176.279,6.749,148.151
C02602=1232.487,306.557,-67.180,-176.277,6.752,148.151
C02603=1232.482,306.805,-67.209,-176.275,6.754,148.151
C02604=1232.478,307.052,-67.239,-176.272,6.757,148.151
C02605=1232.474,307.300,-67.268,-176.270,6.759,148.151
C02606=1232.469,307.549,-67.298,-176.268,6.761,148.151
C02607=1232.465,307.797,-67.328,-176.266,6.764,148.151
C02608=1232.461,308.046,-67.357,-176.264,6.766,148.151
C02609=1232.457,308.294,-67.387,-176.261,6.769,148.151
C02610=1232.453,308.542,-67.417,-176.259,6.771,148.151
C02611=1232.448,308.790,-67.447,-176.257,6.773,148.151
C02612=1232.444,309.038,-67.476,-176.255,6.776,148.151
C02613=1232.439,309.287,-67.506,-176.252,6.779,148.151
C02614=1232.435,309.535,-67.535,-176.250,6.781,148.151
C02615=1232.431,309.783,-67.566,-176.248,6.783,148.151
C02616=1232.427,310.031,-67.596,-176.246,6.785,148.151
C02617=1232.422,310.279,-67.625,-176.243,6.788,148.151
C02618=1232.418,310.528,-67.654,-176.241,6.791,148.150
C02619=1232.414,310.776,-67.685,-176.239,6.793,148.150
C02620=1232.409,311.024,-67.715,-176.237,6.795,148.150
C02621=1232.405,311.272,-67.744,-176.234,6.798,148.150
C02622=1232.401,311.520,-67.774,-176.232,6.800,148.150
C02623=1232.396,311.768,-67.804,-176.230,6.803,148.150
C02624=1232.392,312.017,-67.834,-176.228,6.805,148.150
C02625=1232.388,312.264,-67.864,-176.225,6.808,148.150
C02626=1232.383,312.513,-67.894,-176.223,6.810,148.150
C02627=1232.380,312.761,-67.924,-176.221,6.812,148.150
C02628=1232.375,313.009,-67.954,-176.219,6.815,148.150
C02629=1232.370,313.257,-67.984,-176.216,6.818,148.150
C02630=1232.367,313.505,-68.014,-176.214,6.820,148.150
C02631=1232.362,313.754,-68.044,-176.212,6.822,148.150
C02632=1232.358,314.002,-68.074,-176.210,6.824,148.150
C02633=1232.354,314.250,-68.104,-176.207,6.827,148.150
C02634=1232.350,314.498,-68.135,-176.206,6.830,148.150
C02635=1232.345,314.746,-68.164,-176.204,6.832,148.150
C02636=1232.341,314.995,-68.194,-176.202,6.834,148.150
C02637=1232.336,315.270,-68.228,-176.199,6.837,148.150
C02638=1232.331,315.546,-68.260,-176.196,6.841,148.150
C02639=1232.327,315.822,-68.295,-176.194,6.843,148.150
C02640=1232.322,316.097,-68.327,-176.192,6.846,148.150
C02641=1232.318,316.346,-68.358,-176.189,6.848,148.150
C02642=1232.314,316.594,-68.388,-176.187,6.850,148.150
C02643=1232.309,316.842,-68.419,-176.185,6.853,148.150
C02644=1232.305,317.090,-68.449,-176.183,6.856,148.150
C02645=1232.300,317.338,-68.479,-176.180,6.858,148.150
C02646=1232.296,317.586,-68.509,-176.179,6.860,148.150
C02647=1232.291,317.834,-68.539,-176.176,6.863,148.150
C02648=1232.287,318.082,-68.569,-176.174,6.866,148.150
C02649=1232.283,318.331,-68.600,-176.172,6.868,148.150
C02650=1232.279,318.579,-68.630,-176.169,6.871,148.150
C02651=1232.275,318.827,-68.661,-176.168,6.873,148.150
C02652=1232.271,319.075,-68.691,-176.166,6.876,148.150
C02653=1232.266,319.323,-68.721,-176.164,6.878,148.150
C02654=1232.262,319.571,-68.751,-176.161,6.881,148.150
C02655=1232.257,319.819,-68.782,-176.159,6.883,148.150
C02656=1232.254,320.068,-68.812,-176.157,6.886,148.150
C02657=1232.249,320.316,-68.842,-176.155,6.888,148.150
C02658=1232.245,320.563,-68.872,-176.152,6.891,148.150
C02659=1232.241,320.811,-68.903,-176.150,6.893,148.150
C02660=1232.237,321.060,-68.933,-176.148,6.895,148.150
C02661=1232.233,321.308,-68.964,-176.147,6.898,148.150
C02662=1232.228,321.556,-68.995,-176.144,6.901,148.150
C02663=1232.224,321.804,-69.025,-176.142,6.903,148.150
C02664=1232.219,322.052,-69.056,-176.140,6.906,148.150
C02665=1232.215,322.300,-69.085,-176.138,6.908,148.150
C02666=1232.211,322.549,-69.116,-176.136,6.911,148.150
C02667=1232.207,322.797,-69.147,-176.133,6.913,148.150
C02668=1232.203,323.044,-69.177,-176.131,6.916,148.150
C02669=1232.198,323.292,-69.208,-176.130,6.918,148.150
C02670=1232.194,323.541,-69.239,-176.127,6.921,148.150
C02671=1232.190,323.789,-69.268,-176.125,6.923,148.150
C02672=1232.185,324.037,-69.299,-176.123,6.926,148.150
C02673=1232.181,324.285,-69.329,-176.121,6.928,148.150
C02674=1232.177,324.533,-69.360,-176.119,6.931,148.150
C02675=1232.173,324.781,-69.391,-176.117,6.934,148.151
C02676=1232.168,325.029,-69.422,-176.115,6.936,148.151
C02677=1232.164,325.277,-69.452,-176.112,6.939,148.151
C02678=1232.160,325.526,-69.483,-176.111,6.942,148.151
C02679=1232.156,325.774,-69.514,-176.109,6.944,148.151
C02680=1232.152,326.021,-69.544,-176.106,6.946,148.151
C02681=1232.147,326.269,-69.575,-176.104,6.949,148.151
C02682=1232.143,326.518,-69.606,-176.102,6.952,148.151
C02683=1232.139,326.766,-69.636,-176.100,6.954,148.151
C02684=1232.135,327.013,-69.667,-176.098,6.956,148.151
C02685=1232.131,327.262,-69.698,-176.096,6.959,148.151
C02686=1232.126,327.510,-69.729,-176.094,6.962,148.151
C02687=1232.121,327.758,-69.760,-176.092,6.964,148.151
C02688=1232.118,328.006,-69.790,-176.090,6.966,148.151
C02689=1232.114,328.254,-69.821,-176.088,6.970,148.151
C02690=1232.109,328.502,-69.852,-176.086,6.972,148.151
C02691=1232.104,328.750,-69.883,-176.084,6.974,148.151
C02692=1232.101,328.999,-69.913,-176.082,6.977,148.151
C02693=1232.096,329.247,-69.944,-176.079,6.980,148.151
C02694=1232.092,329.494,-69.975,-176.078,6.982,148.152
C02695=1232.088,329.743,-70.006,-176.076,6.985,148.152
C02696=1232.084,329.991,-70.037,-176.074,6.987,148.151
C02697=1232.079,330.239,-70.068,-176.071,6.990,148.152
C02698=1232.076,330.487,-70.098,-176.069,6.992,148.152
C02699=1232.071,330.735,-70.129,-176.068,6.995,148.152
C02700=1232.067,330.982,-70.161,-176.066,6.997,148.152
C02701=1232.063,331.231,-70.192,-176.063,7.001,148.152
C02702=1232.058,331.479,-70.223,-176.061,7.003,148.152
C02703=1232.053,331.727,-70.253,-176.060,7.005,148.152
C02704=1232.049,331.975,-70.285,-176.058,7.008,148.152
C02705=1232.045,332.223,-70.316,-176.055,7.011,148.152
C02706=1232.042,332.471,-70.347,-176.053,7.013,148.152
C02707=1232.037,332.719,-70.377,-176.052,7.016,148.153
C02708=1232.033,332.966,-70.409,-176.050,7.018,148.152
C02709=1232.029,333.215,-70.440,-176.047,7.021,148.153
C02710=1232.024,333.463,-70.471,-176.045,7.024,148.153
C02711=1232.020,333.712,-70.502,-176.044,7.026,148.153
C02712=1232.016,333.959,-70.533,-176.042,7.028,148.153
C02713=1232.011,334.207,-70.564,-176.039,7.032,148.153
C02714=1232.007,334.456,-70.595,-176.037,7.034,148.153
C02715=1232.003,334.703,-70.627,-176.036,7.036,148.153
C02716=1231.999,334.952,-70.658,-176.034,7.039,148.153
C02717=1231.995,335.199,-70.689,-176.031,7.042,148.153
C02718=1231.990,335.447,-70.720,-176.030,7.045,148.154
C02719=1231.986,335.696,-70.751,-176.028,7.047,148.154
C02720=1231.982,335.943,-70.783,-176.026,7.049,148.154
C02721=1231.978,336.192,-70.814,-176.023,7.052,148.154
C02722=1231.974,336.439,-70.845,-176.022,7.055,148.154
C02723=1231.969,336.688,-70.876,-176.020,7.058,148.154
C02724=1231.965,336.936,-70.907,-176.018,7.060,148.154
C02725=1231.961,337.184,-70.939,-176.016,7.063,148.154
C02726=1231.957,337.432,-70.970,-176.014,7.065,148.154
C02727=1231.953,337.680,-71.002,-176.012,7.068,148.154
C02728=1231.948,337.928,-71.032,-176.011,7.070,148.155
C02729=1231.944,338.175,-71.064,-176.008,7.073,148.155
C02730=1231.940,338.424,-71.095,-176.006,7.076,148.155
C02731=1231.936,338.671,-71.126,-176.005,7.079,148.155
C02732=1231.932,338.919,-71.158,-176.003,7.081,148.155
C02733=1231.927,339.167,-71.189,-176.001,7.083,148.155
C02734=1231.924,339.415,-71.221,-175.999,7.087,148.155
C02735=1231.919,339.663,-71.252,-175.997,7.089,148.155
C02736=1231.915,339.911,-71.284,-175.995,7.091,148.155
C02737=1231.910,340.159,-71.315,-175.994,7.094,148.156
C02738=1231.906,340.407,-71.347,-175.991,7.097,148.156
C02739=1231.902,340.655,-71.377,-175.989,7.100,148.156
C02740=1231.898,340.903,-71.409,-175.988,7.102,148.156
C02741=1231.894,341.181,-71.445,-175.986,7.105,148.156
C02742=1231.888,341.458,-71.479,-175.983,7.108,148.156
C02743=1231.884,341.736,-71.515,-175.981,7.111,148.156
C02744=1231.880,342.013,-71.551,-175.980,7.114,148.157
C02745=1231.874,342.261,-71.582,-175.977,7.117,148.157
C02746=1231.871,342.510,-71.614,-175.975,7.119,148.157
C02747=1231.866,342.757,-71.645,-175.974,7.122,148.157
C02748=1231.862,343.006,-71.676,-175.972,7.124,148.157
C02749=1231.858,343.253,-71.708,-175.970,7.128,148.157
C02750=1231.854,343.501,-71.740,-175.968,7.130,148.157
C02751=1231.849,343.749,-71.772,-175.966,7.132,148.158
C02752=1231.845,343.997,-71.803,-175.965,7.135,148.158
C02753=1231.841,344.245,-71.834,-175.963,7.137,148.158
C02754=1231.837,344.493,-71.866,-175.961,7.141,148.158
C02755=1231.833,344.741,-71.899,-175.959,7.143,148.158
C02756=1231.828,344.989,-71.930,-175.957,7.146,148.158
C02757=1231.824,345.237,-71.961,-175.955,7.148,148.159
C02758=1231.820,345.484,-71.993,-175.954,7.151,148.159
C02759=1231.816,345.733,-72.025,-175.952,7.154,148.159
C02760=1231.811,345.980,-72.057,-175.950,7.157,148.159
C02761=1231.807,346.229,-72.088,-175.948,7.159,148.159
C02762=1231.803,346.477,-72.120,-175.946,7.161,148.159
C02763=1231.799,346.724,-72.152,-175.945,7.164,148.159
C02764=1231.795,346.972,-72.184,-175.943,7.167,148.160
C02765=1231.791,347.220,-72.216,-175.941,7.170,148.160
C02766=1231.786,347.468,-72.248,-175.939,7.172,148.160
C02767=1231.782,347.716,-72.279,-175.938,7.175,148.160
C02768=1231.778,347.963,-72.311,-175.936,7.177,148.160
C02769=1231.774,348.212,-72.343,-175.934,7.181,148.161
C02770=1231.770,348.460,-72.374,-175.932,7.183,148.161
C02771=1231.765,348.708,-72.406,-175.930,7.186,148.161
C02772=1231.761,348.956,-72.438,-175.929,7.188,148.161
C02773=1231.757,349.204,-72.470,-175.927,7.191,148.161
C02774=1231.752,349.452,-72.502,-175.925,7.193,148.161
C02775=1231.749,349.700,-72.534,-175.923,7.196,148.162
C02776=1231.745,349.948,-72.566,-175.922,7.199,148.162
C02777=1231.740,350.195,-72.598,-175.920,7.202,148.162
C02778=1231.736,350.444,-72.630,-175.918,7.204,148.162
C02779=1231.732,350.692,-72.662,-175.917,7.207,148.162
C02780=1231.727,350.939,-72.694,-175.915,7.210,148.163
C02781=1231.724,351.187,-72.726,-175.913,7.213,148.163
C02782=1231.719,351.436,-72.758,-175.911,7.215,148.163
C02783=1231.715,351.682,-72.790,-175.910,7.218,148.163
C02784=1231.711,351.931,-72.823,-175.908,7.220,148.163
C02785=1231.707,352.179,-72.855,-175.906,7.223,148.163
C02786=1231.703,352.426,-72.886,-175.904,7.226,148.164
C02787=1231.698,352.674,-72.919,-175.903,7.229,148.164
C02788=1231.695,352.922,-72.950,-175.901,7.231,148.164
C02789=1231.690,353.170,-72.982,-175.899,7.234,148.164
C02790=1231.686,353.418,-73.014,-175.898,7.236,148.164
C02791=1231.681,353.666,-73.047,-175.897,7.239,148.165
C02792=1231.678,353.914,-73.079,-175.895,7.242,148.165
C02793=1231.673,354.162,-73.111,-175.893,7.245,148.165
C02794=1231.669,354.410,-73.143,-175.891,7.247,148.165
C02795=1231.665,354.658,-73.176,-175.890,7.250,148.166
C02796=1231.660,354.905,-73.207,-175.888,7.252,148.166
C02797=1231.656,355.153,-73.240,-175.886,7.255,148.166
C02798=1231.653,355.401,-73.272,-175.885,7.258,148.166
C02799=1231.648,355.649,-73.305,-175.883,7.260,148.166
C02800=1231.644,355.897,-73.336,-175.881,7.264,148.167
C02801=1231.639,356.145,-73.369,-175.880,7.266,148.167
C02802=1231.636,356.392,-73.401,-175.878,7.269,148.167
C02803=1231.632,356.641,-73.434,-175.876,7.271,148.167
C02804=1231.627,356.888,-73.465,-175.875,7.274,148.168
C02805=1231.623,357.136,-73.498,-175.873,7.276,148.168
C02806=1231.619,357.384,-73.530,-175.872,7.279,148.168
C02807=1231.615,357.632,-73.562,-175.870,7.282,148.168
C02808=1231.611,357.881,-73.595,-175.869,7.284,148.169
C02809=1231.607,358.127,-73.627,-175.867,7.288,148.169
C02810=1231.602,358.376,-73.660,-175.865,7.290,148.169
C02811=1231.598,358.624,-73.691,-175.864,7.293,148.169
C02812=1231.594,358.871,-73.725,-175.862,7.296,148.170
C02813=1231.590,359.120,-73.757,-175.861,7.298,148.170
C02814=1231.586,359.367,-73.789,-175.859,7.301,148.170
C02815=1231.581,359.615,-73.822,-175.858,7.303,148.170
C02816=1231.578,359.863,-73.853,-175.856,7.306,148.170
C02817=1231.574,360.111,-73.887,-175.855,7.308,148.171
C02818=1231.569,360.359,-73.919,-175.853,7.311,148.171
C02819=1231.565,360.606,-73.951,-175.851,7.315,148.171
C02820=1231.561,360.854,-73.984,-175.850,7.317,148.172
C02821=1231.556,361.102,-74.016,-175.848,7.320,148.172
C02822=1231.553,361.350,-74.049,-175.847,7.323,148.172
C02823=1231.548,361.598,-74.081,-175.845,7.325,148.172
C02824=1231.544,361.846,-74.114,-175.844,7.328,148.172
C02825=1231.540,362.093,-74.146,-175.842,7.330,148.173
C02826=1231.536,362.341,-74.179,-175.841,7.333,148.173
C02827=1231.531,362.589,-74.211,-175.839,7.336,148.173
C02828=1231.528,362.837,-74.244,-175.838,7.338,148.174
C02829=1231.523,363.085,-74.276,-175.836,7.341,148.174
C02830=1231.519,363.333,-74.309,-175.835,7.343,148.174
C02831=1231.515,363.581,-74.342,-175.834,7.346,148.174
C02832=1231.511,363.828,-74.374,-175.832,7.349,148.175
C02833=1231.507,364.076,-74.407,-175.831,7.352,148.175
C02834=1231.502,364.324,-74.440,-175.829,7.354,148.175
C02835=1231.499,364.571,-74.472,-175.827,7.358,148.175
C02836=1231.494,364.820,-74.505,-175.826,7.360,148.176
C02837=1231.490,365.067,-74.538,-175.824,7.363,148.176
C02838=1231.486,365.316,-74.570,-175.823,7.366,148.176
C02839=1231.482,365.563,-74.603,-175.822,7.368,148.177
C02840=1231.478,365.810,-74.636,-175.820,7.371,148.177
C02841=1231.473,366.059,-74.668,-175.819,7.374,148.177
C02842=1231.469,366.306,-74.701,-175.817,7.376,148.177
C02843=1231.465,366.554,-74.734,-175.816,7.379,148.178
C02844=1231.461,366.802,-74.766,-175.814,7.381,148.178
C02845=1231.457,367.082,-74.804,-175.813,7.384,148.178
C02846=1231.452,367.361,-74.841,-175.812,7.387,148.179
C02847=1231.447,367.640,-74.877,-175.810,7.391,148.179
C02848=1231.443,367.920,-74.915,-175.809,7.393,148.179
C02849=1231.439,368.168,-74.948,-175.807,7.396,148.180
C02850=1231.434,368.416,-74.980,-175.806,7.399,148.180
C02851=1231.430,368.664,-75.013,-175.804,7.401,148.180
C02852=1231.426,368.911,-75.046,-175.803,7.404,148.181
C02853=1231.422,369.158,-75.079,-175.802,7.407,148.181
C02854=1231.417,369.407,-75.111,-175.800,7.409,148.181
C02855=1231.413,369.654,-75.144,-175.799,7.412,148.182
C02856=1231.409,369.902,-75.178,-175.798,7.415,148.182
C02857=1231.405,370.150,-75.211,-175.796,7.418,148.182
C02858=1231.401,370.398,-75.243,-175.795,7.420,148.182
C02859=1231.397,370.646,-75.276,-175.794,7.423,148.183
C02860=1231.393,370.893,-75.309,-175.792,7.426,148.183
C02861=1231.389,371.141,-75.342,-175.791,7.428,148.183
C02862=1231.385,371.389,-75.375,-175.790,7.431,148.184
C02863=1231.380,371.637,-75.408,-175.788,7.434,148.184
C02864=1231.376,371.885,-75.441,-175.787,7.436,148.184
C02865=1231.372,372.133,-75.474,-175.786,7.438,148.185
C02866=1231.368,372.380,-75.507,-175.785,7.441,148.185
C02867=1231.364,372.628,-75.540,-175.784,7.444,148.185
C02868=1231.360,372.876,-75.573,-175.782,7.447,148.186
C02869=1231.355,373.124,-75.607,-175.781,7.449,148.186
C02870=1231.351,373.371,-75.640,-175.780,7.452,148.186
C02871=1231.348,373.619,-75.672,-175.778,7.455,148.187
C02872=1231.344,373.867,-75.705,-175.777,7.457,148.187
C02873=1231.339,374.115,-75.738,-175.776,7.460,148.187
C02874=1231.335,374.362,-75.771,-175.775,7.462,148.188
C02875=1231.331,374.610,-75.804,-175.774,7.465,148.188
C02876=1231.327,374.858,-75.837,-175.772,7.468,148.188
C02877=1231.323,375.106,-75.871,-175.771,7.470,148.189
C02878=1231.319,375.353,-75.904,-175.770,7.473,148.189
C02879=1231.315,375.601,-75.937,-175.769,7.476,148.189
C02880=1231.310,375.849,-75.970,-175.767,7.479,148.190
C02881=1231.306,376.097,-76.003,-175.767,7.481,148.190
C02882=1231.302,376.344,-76.036,-175.765,7.483,148.190
C02883=1231.298,376.592,-76.069,-175.764,7.486,148.191
C02884=1231.294,376.840,-76.103,-175.763,7.489,148.191
C02885=1231.290,377.088,-76.136,-175.761,7.492,148.191
C02886=1231.286,377.335,-76.169,-175.760,7.494,148.192
C02887=1231.281,377.583,-76.202,-175.760,7.496,148.192
C02888=1231.277,377.831,-76.235,-175.758,7.499,148.192
C02889=1231.272,378.079,-76.269,-175.757,7.502,148.193
C02890=1231.268,378.326,-76.302,-175.756,7.505,148.193
C02891=1231.264,378.574,-76.335,-175.755,7.507,148.193
C02892=1231.261,378.823,-76.369,-175.754,7.509,148.194
C02893=1231.256,379.070,-76.402,-175.753,7.512,148.194
C02894=1231.253,379.317,-76.436,-175.752,7.515,148.195
C02895=1231.249,379.565,-76.469,-175.750,7.518,148.195
C02896=1231.244,379.813,-76.502,-175.749,7.520,148.195
C02897=1231.240,380.061,-76.535,-175.748,7.522,148.195
C02898=1231.236,380.308,-76.568,-175.747,7.525,148.196
C02899=1231.232,380.556,-76.602,-175.746,7.528,148.196
C02900=1231.228,380.804,-76.635,-175.745,7.530,148.197
C02901=1231.223,381.052,-76.669,-175.744,7.533,148.197
C02902=1231.219,381.299,-76.702,-175.743,7.536,148.197
C02903=1231.215,381.547,-76.736,-175.741,7.538,148.198
C02904=1231.211,381.794,-76.769,-175.741,7.540,148.198
C02905=1231.207,382.043,-76.802,-175.739,7.543,148.198
C02906=1231.203,382.291,-76.835,-175.738,7.546,148.199
C02907=1231.199,382.538,-76.869,-175.737,7.549,148.199
C02908=1231.195,382.785,-76.902,-175.737,7.551,148.200
C02909=1231.190,383.033,-76.936,-175.735,7.553,148.200
C02910=1231.186,383.281,-76.969,-175.734,7.556,148.200
C02911=1231.182,383.529,-77.002,-175.734,7.558,148.201
C02912=1231.178,383.776,-77.036,-175.732,7.561,148.201
C02913=1231.174,384.024,-77.069,-175.731,7.564,148.201
C02914=1231.171,384.272,-77.103,-175.730,7.567,148.202
C02915=1231.166,384.520,-77.137,-175.729,7.569,148.202
C02916=1231.162,384.767,-77.171,-175.728,7.572,148.203
C02917=1231.158,385.015,-77.204,-175.727,7.574,148.203
C02918=1231.154,385.263,-77.237,-175.727,7.576,148.203
C02919=1231.150,385.510,-77.271,-175.725,7.579,148.204
C02920=1231.145,385.758,-77.305,-175.724,7.582,148.204
C02921=1231.141,386.006,-77.338,-175.724,7.584,148.204
C02922=1231.137,386.254,-77.371,-175.722,7.587,148.205
C02923=1231.133,386.501,-77.405,-175.721,7.590,148.205
C02924=1231.128,386.749,-77.439,-175.721,7.592,148.206
C02925=1231.124,386.997,-77.472,-175.719,7.594,148.206
C02926=1231.120,387.244,-77.506,-175.719,7.596,148.206
C02927=1231.117,387.493,-77.539,-175.718,7.599,148.207
C02928=1231.113,387.740,-77.573,-175.717,7.602,148.207
C02929=1231.108,387.988,-77.607,-175.716,7.604,148.208
C02930=1231.104,388.235,-77.640,-175.715,7.607,148.208
C02931=1231.100,388.483,-77.674,-175.714,7.610,148.208
C02932=1231.096,388.730,-77.707,-175.713,7.612,148.209
C02933=1231.092,388.979,-77.741,-175.712,7.615,148.209
C02934=1231.088,389.226,-77.775,-175.711,7.616,148.209
C02935=1231.084,389.474,-77.808,-175.710,7.619,148.210
C02936=1231.079,389.721,-77.843,-175.709,7.621,148.210
C02937=1231.075,389.969,-77.876,-175.708,7.624,148.211
C02938=1231.072,390.217,-77.910,-175.707,7.627,148.211
C02939=1231.068,390.465,-77.943,-175.706,7.629,148.211
C02940=1231.063,390.712,-77.978,-175.705,7.632,148.212
C02941=1231.059,390.960,-78.011,-175.705,7.634,148.212
C02942=1231.055,391.207,-78.044,-175.704,7.637,148.213
C02943=1231.051,391.456,-78.079,-175.703,7.639,148.213
C02944=1231.047,391.703,-78.112,-175.702,7.642,148.213
C02945=1231.043,391.950,-78.146,-175.702,7.644,148.214
C02946=1231.038,392.198,-78.180,-175.700,7.646,148.214
C02947=1231.034,392.446,-78.214,-175.699,7.649,148.215
C02948=1231.031,392.694,-78.247,-175.699,7.651,148.215
C02949=1231.026,392.975,-78.286,-175.698,7.654,148.216
C02950=1231.022,393.257,-78.324,-175.697,7.657,148.216
C02951=1231.016,393.537,-78.363,-175.696,7.660,148.216
C02952=1231.012,393.819,-78.402,-175.695,7.662,148.217
C02953=1231.008,394.066,-78.435,-175.694,7.665,148.217
C02954=1231.004,394.314,-78.469,-175.694,7.667,148.218
C02955=1230.999,394.562,-78.503,-175.692,7.670,148.218
C02956=1230.996,394.809,-78.537,-175.692,7.672,148.218
C02957=1230.991,395.057,-78.571,-175.691,7.675,148.219
C02958=1230.987,395.305,-78.604,-175.690,7.677,148.219
C02959=1230.983,395.552,-78.638,-175.689,7.680,148.219
C02960=1230.979,395.800,-78.672,-175.688,7.682,148.220
C02961=1230.975,396.048,-78.706,-175.687,7.685,148.220
C02962=1230.971,396.295,-78.739,-175.687,7.687,148.221
C02963=1230.967,396.543,-78.774,-175.686,7.689,148.221
C02964=1230.963,396.791,-78.808,-175.685,7.691,148.222
C02965=1230.958,397.039,-78.842,-175.684,7.694,148.222
C02966=1230.955,397.286,-78.876,-175.683,7.696,148.222
C02967=1230.950,397.533,-78.910,-175.683,7.699,148.223
C02968=1230.946,397.782,-78.944,-175.682,7.701,148.223
C02969=1230.943,398.029,-78.978,-175.681,7.703,148.224
C02970=1230.938,398.276,-79.012,-175.680,7.706,148.224
C02971=1230.935,398.524,-79.046,-175.680,7.708,148.224
C02972=1230.930,398.772,-79.080,-175.679,7.710,148.225
C02973=1230.926,399.019,-79.114,-175.678,7.713,148.225
C02974=1230.921,399.267,-79.148,-175.678,7.715,148.226
C02975=1230.918,399.515,-79.182,-175.676,7.718,148.226
C02976=1230.913,399.762,-79.216,-175.676,7.720,148.226
C02977=1230.909,400.010,-79.250,-175.676,7.722,148.227
C02978=1230.905,400.258,-79.284,-175.674,7.725,148.227
C02979=1230.902,400.505,-79.318,-175.674,7.727,148.228
C02980=1230.898,400.752,-79.352,-175.673,7.730,148.228
C02981=1230.893,401.001,-79.386,-175.672,7.732,148.228
C02982=1230.890,401.248,-79.420,-175.672,7.734,148.229
C02983=1230.885,401.496,-79.455,-175.671,7.737,148.229
C02984=1230.881,401.743,-79.488,-175.670,7.739,148.230
C02985=1230.877,401.991,-79.523,-175.669,7.741,148.230
C02986=1230.873,402.239,-79.556,-175.668,7.744,148.230
C02987=1230.869,402.486,-79.591,-175.668,7.746,148.231
C02988=1230.865,402.734,-79.625,-175.667,7.748,148.231
C02989=1230.861,402.981,-79.660,-175.666,7.751,148.232
C02990=1230.857,403.229,-79.693,-175.666,7.753,148.232
C02991=1230.853,403.477,-79.728,-175.665,7.755,148.232
C02992=1230.848,403.724,-79.762,-175.664,7.758,148.233
C02993=1230.844,403.972,-79.796,-175.664,7.760,148.233
C02994=1230.840,404.220,-79.831,-175.663,7.762,148.234
C02995=1230.836,404.467,-79.864,-175.662,7.765,148.234
C02996=1230.832,404.715,-79.898,-175.662,7.767,148.235
C02997=1230.828,404.963,-79.933,-175.661,7.769,148.235
C02998=1230.824,405.210,-79.967,-175.660,7.771,148.235
C02999=1230.820,405.457,-80.001,-175.659,7.774,148.236
C03000=1230.816,405.705,-80.036,-175.659,7.776,148.236
C03001=1230.812,405.952,-80.070,-175.658,7.778,148.237
C03002=1230.807,406.200,-80.103,-175.657,7.781,148.237
C03003=1230.803,406.449,-80.138,-175.657,7.783,148.237
C03004=1230.799,406.696,-80.172,-175.656,7.785,148.238
C03005=1230.795,406.944,-80.207,-175.656,7.787,148.238
C03006=1230.792,407.191,-80.241,-175.655,7.790,148.239
C03007=1230.787,407.438,-80.275,-175.654,7.792,148.239
C03008=1230.783,407.686,-80.310,-175.653,7.794,148.239
C03009=1230.779,407.934,-80.344,-175.653,7.796,148.240
C03010=1230.775,408.181,-80.378,-175.652,7.799,148.240
C03011=1230.771,408.429,-80.413,-175.651,7.801,148.241
C03012=1230.767,408.676,-80.447,-175.651,7.803,148.241
C03013=1230.763,408.925,-80.481,-175.651,7.805,148.241
C03014=1230.759,409.172,-80.515,-175.650,7.807,148.242
C03015=1230.754,409.419,-80.550,-175.649,7.810,148.242
C03016=1230.751,409.667,-80.584,-175.648,7.812,148.243
C03017=1230.746,409.915,-80.618,-175.648,7.814,148.243
C03018=1230.742,410.162,-80.653,-175.647,7.816,148.243
C03019=1230.739,410.410,-80.687,-175.646,7.819,148.244
C03020=1230.734,410.657,-80.721,-175.646,7.821,148.244
C03021=1230.731,410.905,-80.756,-175.645,7.823,148.245
C03022=1230.726,411.153,-80.790,-175.645,7.825,148.245
C03023=1230.722,411.400,-80.825,-175.644,7.827,148.245
C03024=1230.718,411.648,-80.859,-175.643,7.830,148.246
C03025=1230.714,411.895,-80.893,-175.643,7.832,148.246
C03026=1230.710,412.143,-80.928,-175.642,7.834,148.247
C03027=1230.706,412.390,-80.962,-175.642,7.836,148.247
C03028=1230.702,412.639,-80.997,-175.641,7.838,148.247
C03029=1230.698,412.886,-81.031,-175.640,7.840,148.248
C03030=1230.694,413.133,-81.065,-175.640,7.843,148.248
C03031=1230.690,413.381,-81.100,-175.639,7.845,148.249
C03032=1230.685,413.628,-81.135,-175.638,7.847,148.249
C03033=1230.682,413.876,-81.169,-175.638,7.849,148.249
C03034=1230.678,414.123,-81.204,-175.638,7.852,148.250
C03035=1230.673,414.371,-81.238,-175.637,7.854,148.250
C03036=1230.669,414.619,-81.273,-175.636,7.856,148.251
C03037=1230.665,414.866,-81.307,-175.635,7.858,148.251
C03038=1230.661,415.114,-81.342,-175.635,7.861,148.252
C03039=1230.657,415.361,-81.376,-175.634,7.863,148.252
C03040=1230.654,415.609,-81.411,-175.634,7.865,148.252
C03041=1230.647,415.981,-81.463,-175.633,7.868,148.253
C03042=1230.641,416.353,-81.515,-175.632,7.871,148.253
C03043=1230.635,416.725,-81.567,-175.631,7.875,148.254
C03044=1230.629,417.096,-81.618,-175.630,7.878,148.255
C03045=1230.208,417.096,-81.651,-175.633,7.888,148.258
C03046=1230.212,416.721,-81.599,-175.635,7.884,148.258
C03047=1230.219,416.348,-81.546,-175.635,7.881,148.257
C03048=1230.225,415.973,-81.494,-175.636,7.878,148.256
C03049=1230.232,415.599,-81.442,-175.637,7.875,148.256
C03050=1230.235,415.351,-81.407,-175.637,7.873,148.255
C03051=1230.239,415.103,-81.373,-175.638,7.871,148.255
C03052=1230.243,414.855,-81.338,-175.639,7.868,148.255
C03053=1230.247,414.608,-81.304,-175.640,7.866,148.254
C03054=1230.252,414.361,-81.270,-175.640,7.864,148.254
C03055=1230.256,414.113,-81.235,-175.641,7.862,148.254
C03056=1230.260,413.866,-81.201,-175.641,7.860,148.253
C03057=1230.263,413.618,-81.165,-175.642,7.858,148.253
C03058=1230.268,413.371,-81.131,-175.642,7.856,148.252
C03059=1230.272,413.123,-81.096,-175.643,7.853,148.252
C03060=1230.276,412.875,-81.062,-175.644,7.851,148.252
C03061=1230.280,412.628,-81.028,-175.645,7.849,148.251
C03062=1230.284,412.380,-80.993,-175.645,7.847,148.251
C03063=1230.288,412.133,-80.959,-175.645,7.845,148.250
C03064=1230.292,411.885,-80.924,-175.646,7.843,148.250
C03065=1230.296,411.637,-80.890,-175.647,7.840,148.250
C03066=1230.300,411.389,-80.856,-175.647,7.838,148.249
C03067=1230.304,411.142,-80.821,-175.648,7.836,148.249
C03068=1230.308,410.895,-80.787,-175.649,7.834,148.248
C03069=1230.312,410.647,-80.752,-175.649,7.832,148.248
C03070=1230.317,410.399,-80.718,-175.650,7.829,148.247
C03071=1230.320,410.152,-80.684,-175.651,7.827,148.247
C03072=1230.324,409.904,-80.649,-175.651,7.825,148.247
C03073=1230.329,409.657,-80.615,-175.652,7.823,148.246
C03074=1230.332,409.409,-80.581,-175.652,7.820,148.246
C03075=1230.337,409.161,-80.546,-175.653,7.817,148.245
C03076=1230.341,408.914,-80.512,-175.654,7.816,148.245
C03077=1230.345,408.666,-80.477,-175.654,7.814,148.245
C03078=1230.349,408.419,-80.443,-175.655,7.811,148.244
C03079=1230.352,408.171,-80.409,-175.656,7.808,148.244
C03080=1230.357,407.924,-80.374,-175.656,7.806,148.243
C03081=1230.362,407.676,-80.340,-175.657,7.804,148.243
C03082=1230.365,407.428,-80.306,-175.657,7.802,148.243
C03083=1230.370,407.180,-80.272,-175.658,7.800,148.242
C03084=1230.373,406.933,-80.238,-175.659,7.797,148.242
C03085=1230.377,406.685,-80.203,-175.660,7.795,148.241
C03086=1230.381,406.438,-80.169,-175.660,7.793,148.241
C03087=1230.385,406.190,-80.134,-175.661,7.790,148.241
C03088=1230.390,405.942,-80.100,-175.662,7.788,148.240
C03089=1230.394,405.695,-80.066,-175.662,7.786,148.240
C03090=1230.398,405.447,-80.031,-175.662,7.784,148.239
C03091=1230.401,405.200,-79.997,-175.664,7.781,148.239
C03092=1230.406,404.952,-79.964,-175.664,7.779,148.239
C03093=1230.410,404.704,-79.929,-175.665,7.777,148.238
C03094=1230.414,404.457,-79.895,-175.666,7.774,148.238
C03095=1230.419,404.209,-79.860,-175.666,7.772,148.237
C03096=1230.422,403.962,-79.826,-175.667,7.770,148.237
C03097=1230.427,403.714,-79.792,-175.667,7.768,148.237
C03098=1230.431,403.466,-79.759,-175.669,7.765,148.236
C03099=1230.435,403.218,-79.724,-175.669,7.763,148.236
C03100=1230.438,402.971,-79.690,-175.669,7.761,148.235
C03101=1230.443,402.724,-79.655,-175.671,7.758,148.235
C03102=1230.446,402.476,-79.621,-175.671,7.756,148.235
C03103=1230.451,402.228,-79.587,-175.671,7.754,148.234
C03104=1230.455,401.981,-79.554,-175.673,7.751,148.234
C03105=1230.459,401.733,-79.519,-175.673,7.749,148.233
C03106=1230.463,401.486,-79.485,-175.674,7.747,148.233
C03107=1230.467,401.238,-79.450,-175.675,7.744,148.233
C03108=1230.471,400.990,-79.417,-175.675,7.742,148.232
C03109=1230.475,400.742,-79.382,-175.676,7.739,148.232
C03110=1230.479,400.495,-79.348,-175.677,7.737,148.231
C03111=1230.483,400.247,-79.314,-175.678,7.735,148.231
C03112=1230.487,399.999,-79.281,-175.678,7.732,148.230
C03113=1230.492,399.752,-79.246,-175.679,7.730,148.230
C03114=1230.496,399.505,-79.212,-175.680,7.728,148.230
C03115=1230.500,399.256,-79.178,-175.681,7.726,148.229
C03116=1230.504,399.009,-79.144,-175.681,7.724,148.229
C03117=1230.508,398.762,-79.110,-175.682,7.720,148.228
C03118=1230.512,398.513,-79.076,-175.683,7.718,148.228
C03119=1230.516,398.266,-79.042,-175.683,7.716,148.228
C03120=1230.520,398.019,-79.008,-175.684,7.714,148.227
C03121=1230.524,397.772,-78.974,-175.685,7.712,148.227
C03122=1230.528,397.523,-78.940,-175.686,7.709,148.226
C03123=1230.532,397.276,-78.906,-175.686,7.707,148.226
C03124=1230.537,397.028,-78.872,-175.688,7.704,148.225
C03125=1230.540,396.780,-78.838,-175.688,7.702,148.225
C03126=1230.544,396.533,-78.804,-175.689,7.700,148.225
C03127=1230.549,396.285,-78.770,-175.690,7.697,148.224
C03128=1230.553,396.038,-78.737,-175.690,7.695,148.224
C03129=1230.557,395.789,-78.702,-175.691,7.692,148.223
C03130=1230.561,395.542,-78.669,-175.692,7.690,148.223
C03131=1230.565,395.295,-78.635,-175.693,7.687,148.223
C03132=1230.570,395.047,-78.601,-175.694,7.685,148.222
C03133=1230.573,394.799,-78.567,-175.695,7.682,148.222
C03134=1230.578,394.551,-78.532,-175.695,7.680,148.221
C03135=1230.582,394.304,-78.499,-175.696,7.677,148.221
C03136=1230.586,394.057,-78.465,-175.697,7.675,148.221
C03137=1230.590,393.808,-78.431,-175.698,7.672,148.220
C03138=1230.595,393.527,-78.393,-175.699,7.670,148.220
C03139=1230.599,393.245,-78.354,-175.699,7.667,148.219
C03140=1230.604,392.965,-78.316,-175.701,7.664,148.219
C03141=1230.608,392.683,-78.278,-175.702,7.662,148.219
C03142=1230.613,392.435,-78.243,-175.703,7.659,148.218
C03143=1230.617,392.188,-78.209,-175.703,7.657,148.218
C03144=1230.621,391.940,-78.176,-175.705,7.654,148.217
C03145=1230.624,391.693,-78.142,-175.705,7.652,148.217
C03146=1230.629,391.445,-78.108,-175.706,7.649,148.216
C03147=1230.633,391.197,-78.074,-175.707,7.647,148.216
C03148=1230.637,390.950,-78.041,-175.708,7.644,148.216
C03149=1230.642,390.702,-78.008,-175.708,7.642,148.215
C03150=1230.645,390.454,-77.973,-175.710,7.639,148.215
C03151=1230.649,390.206,-77.940,-175.710,7.637,148.215
C03152=1230.654,389.959,-77.906,-175.711,7.634,148.214
C03153=1230.658,389.711,-77.873,-175.713,7.632,148.214
C03154=1230.662,389.464,-77.839,-175.713,7.630,148.213
C03155=1230.666,389.215,-77.805,-175.714,7.627,148.213
C03156=1230.670,388.968,-77.771,-175.715,7.625,148.213
C03157=1230.674,388.720,-77.737,-175.716,7.622,148.212
C03158=1230.678,388.473,-77.704,-175.717,7.619,148.212
C03159=1230.683,388.225,-77.670,-175.717,7.617,148.211
C03160=1230.686,387.977,-77.636,-175.719,7.614,148.211
C03161=1230.690,387.730,-77.602,-175.719,7.612,148.211
C03162=1230.694,387.482,-77.569,-175.720,7.609,148.210
C03163=1230.699,387.234,-77.536,-175.722,7.606,148.210
C03164=1230.703,386.987,-77.502,-175.722,7.604,148.209
C03165=1230.707,386.739,-77.469,-175.723,7.602,148.209
C03166=1230.710,386.491,-77.435,-175.724,7.599,148.209
C03167=1230.715,386.243,-77.401,-175.725,7.597,148.208
C03168=1230.719,385.995,-77.367,-175.726,7.594,148.208
C03169=1230.723,385.748,-77.334,-175.727,7.591,148.208
C03170=1230.727,385.501,-77.300,-175.728,7.589,148.207
C03171=1230.731,385.253,-77.267,-175.729,7.586,148.207
C03172=1230.736,385.005,-77.233,-175.730,7.584,148.206
C03173=1230.739,384.757,-77.199,-175.731,7.582,148.206
C03174=1230.744,384.509,-77.166,-175.732,7.579,148.206
C03175=1230.748,384.262,-77.133,-175.733,7.576,148.205
C03176=1230.752,384.014,-77.100,-175.734,7.574,148.205
C03177=1230.756,383.766,-77.065,-175.735,7.571,148.204
C03178=1230.760,383.519,-77.032,-175.736,7.568,148.204
C03179=1230.765,383.271,-76.999,-175.737,7.566,148.204
C03180=1230.769,383.023,-76.966,-175.738,7.564,148.203
C03181=1230.772,382.775,-76.932,-175.739,7.561,148.203
C03182=1230.776,382.528,-76.898,-175.740,7.558,148.203
C03183=1230.781,382.280,-76.865,-175.741,7.556,148.202
C03184=1230.785,382.032,-76.832,-175.743,7.553,148.202
C03185=1230.789,381.784,-76.798,-175.744,7.551,148.202
C03186=1230.793,381.537,-76.764,-175.744,7.549,148.201
C03187=1230.797,381.289,-76.731,-175.746,7.546,148.201
C03188=1230.801,381.042,-76.698,-175.747,7.543,148.200
C03189=1230.806,380.794,-76.665,-175.748,7.540,148.200
C03190=1230.810,380.546,-76.632,-175.749,7.538,148.200
C03191=1230.814,380.297,-76.598,-175.750,7.535,148.199
C03192=1230.818,380.050,-76.564,-175.751,7.532,148.199
C03193=1230.822,379.803,-76.531,-175.753,7.530,148.199
C03194=1230.826,379.555,-76.498,-175.754,7.527,148.198
C03195=1230.830,379.307,-76.464,-175.754,7.525,148.198
C03196=1230.834,379.059,-76.431,-175.755,7.522,148.198
C03197=1230.838,378.812,-76.398,-175.757,7.519,148.197
C03198=1230.843,378.564,-76.365,-175.758,7.517,148.197
C03199=1230.847,378.316,-76.332,-175.759,7.514,148.196
C03200=1230.851,378.068,-76.299,-175.760,7.512,148.196
C03201=1230.855,377.821,-76.265,-175.761,7.509,148.196
C03202=1230.859,377.573,-76.232,-175.762,7.506,148.195
C03203=1230.863,377.325,-76.199,-175.764,7.504,148.195
C03204=1230.867,377.078,-76.165,-175.765,7.501,148.195
C03205=1230.871,376.830,-76.132,-175.766,7.499,148.195
C03206=1230.876,376.582,-76.098,-175.767,7.496,148.194
C03207=1230.880,376.334,-76.065,-175.768,7.493,148.194
C03208=1230.884,376.086,-76.032,-175.769,7.491,148.193
C03209=1230.888,375.838,-75.999,-175.770,7.488,148.193
C03210=1230.892,375.591,-75.965,-175.772,7.485,148.193
C03211=1230.896,375.343,-75.932,-175.773,7.483,148.192
C03212=1230.900,375.095,-75.899,-175.774,7.480,148.192
C03213=1230.905,374.848,-75.866,-175.775,7.478,148.192
C03214=1230.909,374.599,-75.833,-175.777,7.475,148.191
C03215=1230.912,374.352,-75.801,-175.778,7.472,148.191
C03216=1230.916,374.104,-75.768,-175.779,7.469,148.191
C03217=1230.921,373.856,-75.735,-175.781,7.467,148.190
C03218=1230.925,373.609,-75.701,-175.782,7.464,148.190
C03219=1230.929,373.361,-75.668,-175.782,7.462,148.190
C03220=1230.933,373.113,-75.635,-175.783,7.459,148.189
C03221=1230.937,372.865,-75.602,-175.785,7.457,148.189
C03222=1230.941,372.618,-75.569,-175.786,7.454,148.189
C03223=1230.945,372.370,-75.536,-175.787,7.451,148.188
C03224=1230.950,372.122,-75.503,-175.789,7.449,148.188
C03225=1230.954,371.874,-75.470,-175.790,7.446,148.188
C03226=1230.958,371.626,-75.437,-175.791,7.443,148.187
C03227=1230.962,371.378,-75.404,-175.793,7.440,148.187
C03228=1230.966,371.131,-75.371,-175.794,7.438,148.187
C03229=1230.971,370.883,-75.337,-175.796,7.435,148.187
C03230=1230.975,370.635,-75.304,-175.797,7.432,148.186
C03231=1230.979,370.388,-75.273,-175.798,7.429,148.186
C03232=1230.983,370.140,-75.240,-175.800,7.427,148.186
C03233=1230.987,369.892,-75.207,-175.800,7.425,148.185
C03234=1230.991,369.645,-75.173,-175.802,7.422,148.185
C03235=1230.996,369.397,-75.140,-175.803,7.419,148.185
C03236=1231.000,369.149,-75.108,-175.804,7.417,148.184
C03237=1231.004,368.901,-75.075,-175.806,7.414,148.184
C03238=1231.008,368.653,-75.042,-175.807,7.411,148.184
C03239=1231.012,368.406,-75.009,-175.809,7.409,148.183
C03240=1231.016,368.157,-74.976,-175.810,7.406,148.183
C03241=1231.020,367.910,-74.943,-175.811,7.403,148.183
C03242=1231.025,367.630,-74.906,-175.813,7.400,148.182
C03243=1231.030,367.351,-74.870,-175.814,7.397,148.182
C03244=1231.034,367.071,-74.832,-175.816,7.394,148.182
C03245=1231.039,366.792,-74.795,-175.818,7.391,148.181
C03246=1231.043,366.543,-74.762,-175.819,7.388,148.181
C03247=1231.047,366.296,-74.730,-175.820,7.385,148.181
C03248=1231.051,366.049,-74.697,-175.822,7.383,148.181
C03249=1231.056,365.801,-74.665,-175.823,7.380,148.180
C03250=1231.060,365.553,-74.631,-175.825,7.377,148.180
C03251=1231.064,365.305,-74.600,-175.826,7.375,148.180
C03252=1231.068,365.057,-74.566,-175.828,7.372,148.179
C03253=1231.072,364.809,-74.533,-175.829,7.370,148.179
C03254=1231.076,364.561,-74.501,-175.830,7.367,148.179
C03255=1231.080,364.314,-74.468,-175.832,7.364,148.179
C03256=1231.084,364.065,-74.436,-175.833,7.361,148.178
C03257=1231.089,363.818,-74.403,-175.835,7.359,148.178
C03258=1231.093,363.571,-74.370,-175.836,7.356,148.178
C03259=1231.097,363.322,-74.338,-175.838,7.354,148.177
C03260=1231.101,363.075,-74.305,-175.839,7.351,148.177
C03261=1231.105,362.826,-74.272,-175.840,7.348,148.177
C03262=1231.109,362.579,-74.240,-175.842,7.346,148.177
C03263=1231.113,362.331,-74.207,-175.844,7.342,148.176
C03264=1231.118,362.084,-74.175,-175.845,7.339,148.176
C03265=1231.122,361.835,-74.142,-175.847,7.337,148.176
C03266=1231.126,361.588,-74.110,-175.849,7.334,148.176
C03267=1231.130,361.339,-74.077,-175.850,7.332,148.175
C03268=1231.134,361.092,-74.044,-175.851,7.329,148.175
C03269=1231.138,360.844,-74.012,-175.853,7.326,148.175
C03270=1231.143,360.596,-73.980,-175.855,7.324,148.175
C03271=1231.147,360.349,-73.948,-175.856,7.321,148.174
C03272=1231.151,360.100,-73.915,-175.857,7.319,148.174
C03273=1231.155,359.853,-73.882,-175.859,7.316,148.174
C03274=1231.159,359.605,-73.850,-175.860,7.313,148.174
C03275=1231.163,359.357,-73.817,-175.862,7.310,148.173
C03276=1231.168,359.109,-73.785,-175.864,7.307,148.173
C03277=1231.172,358.861,-73.753,-175.866,7.305,148.173
C03278=1231.176,358.613,-73.720,-175.867,7.302,148.173
C03279=1231.180,358.365,-73.688,-175.868,7.299,148.172
C03280=1231.184,358.117,-73.656,-175.870,7.297,148.172
C03281=1231.189,357.870,-73.623,-175.872,7.294,148.172
C03282=1231.193,357.622,-73.591,-175.873,7.292,148.172
C03283=1231.197,357.374,-73.559,-175.874,7.289,148.171
C03284=1231.200,357.126,-73.526,-175.877,7.286,148.171
C03285=1231.205,356.879,-73.494,-175.878,7.283,148.171
C03286=1231.209,356.630,-73.462,-175.880,7.281,148.171
C03287=1231.214,356.382,-73.430,-175.881,7.278,148.171
C03288=1231.218,356.134,-73.397,-175.883,7.275,148.170
C03289=1231.222,355.887,-73.365,-175.884,7.273,148.170
C03290=1231.226,355.639,-73.333,-175.886,7.270,148.170
C03291=1231.230,355.391,-73.301,-175.888,7.267,148.170
C03292=1231.234,355.143,-73.268,-175.890,7.264,148.169
C03293=1231.239,354.896,-73.236,-175.891,7.262,148.169
C03294=1231.243,354.647,-73.204,-175.893,7.259,148.169
C03295=1231.247,354.399,-73.172,-175.895,7.257,148.169
C03296=1231.251,354.151,-73.139,-175.896,7.254,148.168
C03297=1231.255,353.904,-73.107,-175.897,7.251,148.168
C03298=1231.260,353.656,-73.075,-175.899,7.248,148.168
C03299=1231.263,353.408,-73.043,-175.901,7.245,148.168
C03300=1231.268,353.159,-73.010,-175.903,7.243,148.168
C03301=1231.272,352.912,-72.979,-175.904,7.240,148.167
C03302=1231.277,352.664,-72.947,-175.906,7.238,148.167
C03303=1231.280,352.416,-72.914,-175.908,7.235,148.167
C03304=1231.284,352.169,-72.883,-175.910,7.232,148.167
C03305=1231.289,351.921,-72.850,-175.911,7.229,148.167
C03306=1231.292,351.673,-72.818,-175.913,7.227,148.166
C03307=1231.297,351.425,-72.786,-175.915,7.224,148.166
C03308=1231.301,351.177,-72.754,-175.916,7.222,148.166
C03309=1231.306,350.929,-72.722,-175.918,7.219,148.166
C03310=1231.310,350.681,-72.690,-175.920,7.216,148.166
C03311=1231.314,350.433,-72.659,-175.922,7.213,148.166
C03312=1231.318,350.185,-72.626,-175.923,7.211,148.165
C03313=1231.322,349.937,-72.595,-175.925,7.208,148.165
C03314=1231.327,349.689,-72.562,-175.927,7.206,148.165
C03315=1231.331,349.441,-72.530,-175.928,7.203,148.165
C03316=1231.335,349.194,-72.499,-175.930,7.200,148.165
C03317=1231.339,348.945,-72.466,-175.932,7.197,148.164
C03318=1231.343,348.697,-72.435,-175.934,7.195,148.164
C03319=1231.347,348.450,-72.403,-175.935,7.192,148.164
C03320=1231.352,348.202,-72.371,-175.937,7.190,148.164
C03321=1231.355,347.954,-72.339,-175.939,7.186,148.164
C03322=1231.360,347.706,-72.307,-175.941,7.184,148.163
C03323=1231.364,347.458,-72.275,-175.942,7.181,148.163
C03324=1231.368,347.211,-72.243,-175.944,7.179,148.163
C03325=1231.373,346.962,-72.212,-175.946,7.177,148.163
C03326=1231.377,346.714,-72.180,-175.948,7.173,148.163
C03327=1231.381,346.466,-72.148,-175.950,7.171,148.163
C03328=1231.385,346.218,-72.117,-175.951,7.168,148.162
C03329=1231.389,345.970,-72.085,-175.953,7.166,148.162
C03330=1231.394,345.723,-72.053,-175.955,7.163,148.162
C03331=1231.397,345.474,-72.021,-175.957,7.160,148.162
C03332=1231.402,345.227,-71.990,-175.959,7.157,148.162
C03333=1231.406,344.978,-71.958,-175.960,7.155,148.162
C03334=1231.411,344.731,-71.926,-175.962,7.152,148.162
C03335=1231.414,344.483,-71.894,-175.964,7.150,148.161
C03336=1231.418,344.235,-71.862,-175.966,7.146,148.161
C03337=1231.424,343.986,-71.831,-175.968,7.144,148.161
C03338=1231.427,343.738,-71.799,-175.970,7.142,148.161
C03339=1231.432,343.491,-71.768,-175.971,7.139,148.161
C03340=1231.435,343.243,-71.736,-175.973,7.136,148.161
C03341=1231.440,342.995,-71.705,-175.975,7.133,148.160
C03342=1231.444,342.747,-71.673,-175.977,7.131,148.160
C03343=1231.449,342.499,-71.641,-175.979,7.128,148.160
C03344=1231.453,342.251,-71.610,-175.980,7.126,148.160
C03345=1231.456,342.003,-71.578,-175.983,7.123,148.160
C03346=1231.461,341.726,-71.543,-175.985,7.120,148.160
C03347=1231.466,341.448,-71.508,-175.987,7.117,148.160
C03348=1231.470,341.170,-71.472,-175.988,7.114,148.159
C03349=1231.476,340.893,-71.437,-175.991,7.111,148.159
C03350=1231.480,340.644,-71.405,-175.993,7.109,148.159
C03351=1231.484,340.397,-71.374,-175.995,7.105,148.159
C03352=1231.488,340.148,-71.343,-175.996,7.103,148.159
C03353=1231.493,339.901,-71.311,-175.999,7.101,148.159
C03354=1231.496,339.653,-71.280,-176.000,7.098,148.159
C03355=1231.501,339.405,-71.249,-176.002,7.096,148.159
C03356=1231.505,339.157,-71.217,-176.004,7.093,148.158
C03357=1231.509,338.909,-71.186,-176.006,7.090,148.158
C03358=1231.514,338.661,-71.154,-176.008,7.088,148.158
C03359=1231.518,338.413,-71.123,-176.010,7.085,148.158
C03360=1231.522,338.165,-71.091,-176.012,7.082,148.158
C03361=1231.527,337.917,-71.060,-176.014,7.079,148.158
C03362=1231.530,337.669,-71.029,-176.016,7.077,148.158
C03363=1231.535,337.421,-70.998,-176.017,7.075,148.158
C03364=1231.539,337.173,-70.966,-176.019,7.071,148.157
C03365=1231.543,336.925,-70.935,-176.022,7.069,148.157
C03366=1231.547,336.677,-70.904,-176.023,7.066,148.157
C03367=1231.551,336.429,-70.873,-176.025,7.064,148.157
C03368=1231.556,336.181,-70.841,-176.027,7.061,148.157
C03369=1231.560,335.933,-70.810,-176.029,7.058,148.157
C03370=1231.564,335.685,-70.778,-176.031,7.056,148.157
C03371=1231.568,335.437,-70.747,-176.033,7.054,148.157
C03372=1231.573,335.189,-70.717,-176.035,7.051,148.157
C03373=1231.576,334.941,-70.685,-176.037,7.048,148.157
C03374=1231.581,334.693,-70.654,-176.039,7.046,148.157
C03375=1231.586,334.445,-70.623,-176.041,7.043,148.156
C03376=1231.589,334.197,-70.591,-176.043,7.040,148.156
C03377=1231.594,333.949,-70.561,-176.045,7.038,148.156
C03378=1231.598,333.700,-70.529,-176.047,7.035,148.156
C03379=1231.602,333.453,-70.498,-176.049,7.033,148.156
C03380=1231.607,333.205,-70.467,-176.051,7.029,148.156
C03381=1231.611,332.956,-70.436,-176.053,7.027,148.156
C03382=1231.615,332.709,-70.405,-176.055,7.025,148.156
C03383=1231.619,332.461,-70.374,-176.057,7.023,148.156
C03384=1231.623,332.213,-70.343,-176.059,7.019,148.155
C03385=1231.628,331.965,-70.313,-176.061,7.017,148.156
C03386=1231.631,331.717,-70.281,-176.063,7.014,148.155
C03387=1231.636,331.469,-70.250,-176.065,7.012,148.155
C03388=1231.641,331.221,-70.219,-176.067,7.009,148.155
C03389=1231.645,330.972,-70.188,-176.069,7.007,148.155
C03390=1231.649,330.725,-70.157,-176.071,7.004,148.155
C03391=1231.652,330.476,-70.126,-176.073,7.002,148.155
C03392=1231.657,330.228,-70.095,-176.075,6.998,148.155
C03393=1231.662,329.980,-70.064,-176.077,6.996,148.155
C03394=1231.666,329.732,-70.033,-176.079,6.994,148.155
C03395=1231.670,329.484,-70.003,-176.081,6.991,148.155
C03396=1231.674,329.237,-69.971,-176.083,6.988,148.155
C03397=1231.678,328.988,-69.941,-176.085,6.986,148.155
C03398=1231.682,328.740,-69.910,-176.087,6.984,148.155
C03399=1231.687,328.492,-69.879,-176.089,6.980,148.154
C03400=1231.692,328.244,-69.848,-176.091,6.978,148.154
C03401=1231.696,327.996,-69.817,-176.093,6.976,148.154
C03402=1231.699,327.748,-69.787,-176.095,6.973,148.154
C03403=1231.704,327.500,-69.756,-176.098,6.970,148.154
C03404=1231.708,327.251,-69.725,-176.099,6.968,148.154
C03405=1231.713,327.003,-69.694,-176.101,6.965,148.154
C03406=1231.717,326.756,-69.664,-176.103,6.963,148.154
C03407=1231.721,326.507,-69.633,-176.106,6.960,148.154
C03408=1231.725,326.259,-69.602,-176.108,6.958,148.154
C03409=1231.730,326.011,-69.571,-176.110,6.955,148.154
C03410=1231.734,325.764,-69.541,-176.111,6.953,148.154
C03411=1231.738,325.515,-69.510,-176.114,6.950,148.154
C03412=1231.742,325.267,-69.479,-176.116,6.948,148.154
C03413=1231.746,325.019,-69.449,-176.118,6.945,148.154
C03414=1231.750,324.771,-69.418,-176.120,6.942,148.154
C03415=1231.755,324.523,-69.387,-176.123,6.940,148.154
C03416=1231.759,324.275,-69.357,-176.124,6.937,148.154
C03417=1231.763,324.027,-69.326,-176.126,6.935,148.154
C03418=1231.767,323.778,-69.295,-176.129,6.932,148.154
C03419=1231.771,323.531,-69.265,-176.131,6.929,148.153
C03420=1231.776,323.282,-69.235,-176.133,6.927,148.153
C03421=1231.781,323.034,-69.204,-176.135,6.925,148.154
C03422=1231.785,322.787,-69.174,-176.137,6.922,148.154
C03423=1231.789,322.538,-69.143,-176.139,6.919,148.153
C03424=1231.793,322.290,-69.112,-176.141,6.917,148.153
C03425=1231.797,322.042,-69.082,-176.143,6.915,148.153
C03426=1231.802,321.794,-69.052,-176.146,6.912,148.153
C03427=1231.805,321.545,-69.022,-176.147,6.909,148.153
C03428=1231.810,321.297,-68.991,-176.150,6.907,148.153
C03429=1231.815,321.049,-68.960,-176.152,6.904,148.153
C03430=1231.818,320.802,-68.930,-176.154,6.902,148.153
C03431=1231.823,320.553,-68.900,-176.156,6.899,148.153
C03432=1231.827,320.306,-68.870,-176.158,6.897,148.153
C03433=1231.831,320.057,-68.838,-176.161,6.894,148.153
C03434=1231.835,319.809,-68.808,-176.163,6.892,148.153
C03435=1231.840,319.561,-68.778,-176.165,6.889,148.153
C03436=1231.844,319.313,-68.748,-176.166,6.887,148.153
C03437=1231.848,319.065,-68.717,-176.169,6.884,148.153
C03438=1231.853,318.817,-68.688,-176.171,6.882,148.153
C03439=1231.857,318.568,-68.657,-176.173,6.879,148.153
C03440=1231.861,318.321,-68.627,-176.175,6.877,148.153
C03441=1231.865,318.072,-68.597,-176.178,6.874,148.153
C03442=1231.869,317.824,-68.566,-176.180,6.872,148.153
C03443=1231.874,317.576,-68.536,-176.182,6.869,148.153
C03444=1231.878,317.328,-68.506,-176.184,6.866,148.153
C03445=1231.883,317.080,-68.475,-176.187,6.864,148.153
C03446=1231.886,316.831,-68.446,-176.189,6.862,148.153
C03447=1231.891,316.583,-68.415,-176.190,6.859,148.153
C03448=1231.895,316.335,-68.385,-176.193,6.856,148.153
C03449=1231.900,316.087,-68.355,-176.195,6.854,148.153
C03450=1231.904,315.811,-68.322,-176.197,6.852,148.153
C03451=1231.909,315.536,-68.288,-176.200,6.849,148.153
C03452=1231.914,315.260,-68.255,-176.202,6.846,148.153
C03453=1231.919,314.984,-68.220,-176.204,6.843,148.153
C03454=1231.923,314.736,-68.191,-176.207,6.840,148.153
C03455=1231.927,314.488,-68.161,-176.209,6.838,148.153
C03456=1231.932,314.239,-68.131,-176.211,6.836,148.153
C03457=1231.935,313.992,-68.101,-176.213,6.834,148.153
C03458=1231.940,313.744,-68.071,-176.216,6.831,148.153
C03459=1231.944,313.496,-68.040,-176.218,6.828,148.153
C03460=1231.948,313.247,-68.011,-176.220,6.826,148.153
C03461=1231.953,312.999,-67.981,-176.222,6.824,148.153
C03462=1231.957,312.751,-67.951,-176.225,6.821,148.153
C03463=1231.961,312.503,-67.921,-176.227,6.818,148.153
C03464=1231.966,312.255,-67.890,-176.229,6.816,148.153
C03465=1231.970,312.007,-67.861,-176.231,6.814,148.153
C03466=1231.974,311.758,-67.832,-176.233,6.811,148.153
C03467=1231.979,311.510,-67.801,-176.236,6.809,148.153
C03468=1231.983,311.262,-67.771,-176.238,6.806,148.153
C03469=1231.987,311.014,-67.742,-176.240,6.804,148.154
C03470=1231.991,310.766,-67.712,-176.242,6.801,148.154
C03471=1231.996,310.518,-67.682,-176.245,6.799,148.154
C03472=1232.000,310.269,-67.652,-176.247,6.797,148.154
C03473=1232.004,310.021,-67.623,-176.249,6.794,148.154
C03474=1232.009,309.773,-67.592,-176.251,6.791,148.154
C03475=1232.013,309.525,-67.563,-176.253,6.789,148.154
C03476=1232.017,309.277,-67.533,-176.256,6.787,148.154
C03477=1232.022,309.028,-67.504,-176.258,6.785,148.154
C03478=1232.026,308.780,-67.473,-176.260,6.782,148.154
C03479=1232.030,308.532,-67.443,-176.262,6.779,148.154
C03480=1232.035,308.284,-67.414,-176.265,6.777,148.154
C03481=1232.039,308.036,-67.385,-176.267,6.775,148.154
C03482=1232.043,307.787,-67.355,-176.269,6.772,148.154
C03483=1232.048,307.539,-67.324,-176.271,6.770,148.154
C03484=1232.052,307.291,-67.295,-176.273,6.767,148.154
C03485=1232.056,307.043,-67.265,-176.276,6.765,148.154
C03486=1232.060,306.795,-67.236,-176.278,6.762,148.154
C03487=1232.064,306.546,-67.207,-176.280,6.760,148.154
C03488=1232.069,306.298,-67.177,-176.282,6.758,148.154
C03489=1232.073,306.049,-67.147,-176.285,6.755,148.154
C03490=1232.078,305.801,-67.118,-176.288,6.753,148.155
C03491=1232.081,305.553,-67.087,-176.290,6.750,148.155
C03492=1232.086,305.305,-67.058,-176.292,6.748,148.155
C03493=1232.090,305.058,-67.029,-176.294,6.746,148.155
C03494=1232.095,304.809,-66.999,-176.297,6.743,148.155
C03495=1232.099,304.561,-66.970,-176.299,6.741,148.155
C03496=1232.104,304.313,-66.940,-176.301,6.738,148.155
C03497=1232.108,304.064,-66.910,-176.303,6.736,148.155
C03498=1232.112,303.816,-66.881,-176.306,6.733,148.155
C03499=1232.116,303.568,-66.852,-176.308,6.731,148.155
C03500=1232.120,303.319,-66.822,-176.310,6.729,148.155
C03501=1232.125,303.071,-66.793,-176.312,6.727,148.155
C03502=1232.129,302.823,-66.763,-176.314,6.725,148.155
C03503=1232.134,302.575,-66.734,-176.317,6.722,148.155
C03504=1232.138,302.327,-66.705,-176.319,6.719,148.155
C03505=1232.142,302.078,-66.676,-176.321,6.717,148.155
C03506=1232.146,301.830,-66.646,-176.323,6.715,148.155
C03507=1232.151,301.582,-66.617,-176.326,6.712,148.155
C03508=1232.155,301.333,-66.588,-176.329,6.710,148.156
C03509=1232.159,301.085,-66.558,-176.331,6.708,148.156
C03510=1232.164,300.838,-66.529,-176.333,6.705,148.156
C03511=1232.168,300.589,-66.500,-176.336,6.702,148.156
C03512=1232.172,300.341,-66.470,-176.338,6.700,148.156
C03513=1232.177,300.092,-66.441,-176.340,6.698,148.156
C03514=1232.181,299.844,-66.412,-176.342,6.696,148.156
C03515=1232.185,299.596,-66.382,-176.344,6.694,148.156
C03516=1232.190,299.348,-66.353,-176.347,6.691,148.156
C03517=1232.194,299.100,-66.324,-176.349,6.689,148.156
C03518=1232.198,298.851,-66.295,-176.351,6.686,148.156
C03519=1232.203,298.603,-66.266,-176.353,6.684,148.157
C03520=1232.207,298.354,-66.236,-176.357,6.681,148.157
C03521=1232.212,298.107,-66.207,-176.359,6.679,148.157
C03522=1232.216,297.858,-66.178,-176.361,6.677,148.157
C03523=1232.220,297.610,-66.149,-176.363,6.675,148.157
C03524=1232.224,297.362,-66.120,-176.365,6.673,148.157
C03525=1232.229,297.113,-66.092,-176.368,6.670,148.157
C03526=1232.233,296.865,-66.062,-176.370,6.667,148.157
C03527=1232.237,296.617,-66.033,-176.372,6.665,148.157
C03528=1232.242,296.368,-66.004,-176.374,6.663,148.157
C03529=1232.246,296.120,-65.975,-176.377,6.661,148.158
C03530=1232.251,295.872,-65.946,-176.380,6.658,148.158
C03531=1232.254,295.624,-65.917,-176.382,6.656,148.158
C03532=1232.259,295.375,-65.888,-176.384,6.654,148.158
C03533=1232.263,295.127,-65.859,-176.386,6.652,148.158
C03534=1232.268,294.879,-65.830,-176.389,6.649,148.158
C03535=1232.272,294.631,-65.801,-176.391,6.646,148.158
C03536=1232.276,294.382,-65.772,-176.393,6.644,148.158
C03537=1232.280,294.134,-65.743,-176.396,6.642,148.158
C03538=1232.285,293.886,-65.714,-176.398,6.640,148.159
C03539=1232.289,293.637,-65.685,-176.400,6.638,148.159
C03540=1232.293,293.389,-65.656,-176.403,6.635,148.159
C03541=1232.298,293.141,-65.628,-176.405,6.633,148.159
C03542=1232.302,292.893,-65.599,-176.407,6.631,148.159
C03543=1232.306,292.644,-65.570,-176.410,6.628,148.159
C03544=1232.311,292.397,-65.541,-176.412,6.627,148.159
C03545=1232.315,292.148,-65.513,-176.415,6.623,148.159
C03546=1232.319,291.899,-65.484,-176.417,6.621,148.159
C03547=1232.324,291.651,-65.454,-176.419,6.619,148.160
C03548=1232.329,291.403,-65.426,-176.422,6.617,148.160
C03549=1232.332,291.155,-65.397,-176.424,6.615,148.160
C03550=1232.337,290.906,-65.368,-176.427,6.612,148.160
C03551=1232.341,290.658,-65.339,-176.429,6.610,148.160
C03552=1232.345,290.410,-65.311,-176.431,6.608,148.160
C03553=1232.350,290.161,-65.282,-176.434,6.606,148.160
C03554=1232.355,289.888,-65.250,-176.436,6.603,148.160
C03555=1232.360,289.613,-65.219,-176.439,6.601,148.161
C03556=1232.364,289.339,-65.187,-176.441,6.598,148.161
C03557=1232.369,289.065,-65.156,-176.444,6.596,148.161
C03558=1232.373,288.817,-65.127,-176.446,6.594,148.161
C03559=1232.378,288.568,-65.098,-176.449,6.591,148.161
C03560=1232.383,288.320,-65.070,-176.451,6.589,148.161
C03561=1232.387,288.072,-65.042,-176.454,6.586,148.161
C03562=1232.391,287.823,-65.012,-176.456,6.584,148.161
C03563=1232.395,287.576,-64.985,-176.458,6.582,148.162
C03564=1232.400,287.327,-64.956,-176.460,6.580,148.162
C03565=1232.404,287.078,-64.927,-176.463,6.577,148.162
C03566=1232.408,286.831,-64.899,-176.466,6.575,148.162
C03567=1232.413,286.582,-64.870,-176.468,6.573,148.162
C03568=1232.417,286.334,-64.842,-176.470,6.571,148.162
C03569=1232.421,286.085,-64.813,-176.472,6.569,148.163
C03570=1232.426,285.837,-64.785,-176.475,6.567,148.163
C03571=1232.430,285.589,-64.756,-176.478,6.564,148.163
C03572=1232.434,285.340,-64.727,-176.480,6.562,148.163
C03573=1232.439,285.092,-64.700,-176.482,6.560,148.163
C03574=1232.443,284.843,-64.671,-176.484,6.557,148.163
C03575=1232.448,284.595,-64.643,-176.487,6.555,148.163
C03576=1232.452,284.346,-64.614,-176.489,6.553,148.164
C03577=1232.456,284.098,-64.587,-176.491,6.551,148.164
C03578=1232.461,283.850,-64.557,-176.494,6.548,148.164
C03579=1232.465,283.602,-64.529,-176.497,6.546,148.164
C03580=1232.469,283.353,-64.501,-176.499,6.544,148.164
C03581=1232.474,283.106,-64.473,-176.501,6.542,148.164
C03582=1232.478,282.857,-64.444,-176.503,6.540,148.164
C03583=1232.482,282.608,-64.416,-176.506,6.538,148.165
C03584=1232.487,282.360,-64.388,-176.509,6.535,148.165
C03585=1232.491,282.111,-64.359,-176.511,6.533,148.165
C03586=1232.495,281.863,-64.332,-176.513,6.531,148.165
C03587=1232.500,281.615,-64.303,-176.516,6.529,148.165
C03588=1232.504,281.367,-64.275,-176.518,6.527,148.165
C03589=1232.509,281.118,-64.246,-176.520,6.524,148.165
C03590=1232.513,280.870,-64.219,-176.523,6.522,148.166
C03591=1232.517,280.621,-64.190,-176.525,6.520,148.166
C03592=1232.522,280.373,-64.162,-176.528,6.518,148.166
C03593=1232.525,280.125,-64.134,-176.530,6.515,148.166
C03594=1232.531,279.876,-64.106,-176.533,6.513,148.166
C03595=1232.535,279.628,-64.079,-176.535,6.511,148.166
C03596=1232.539,279.379,-64.050,-176.537,6.509,148.167
C03597=1232.544,279.131,-64.022,-176.539,6.507,148.167
C03598=1232.548,278.883,-63.994,-176.542,6.505,148.167
C03599=1232.552,278.635,-63.966,-176.545,6.502,148.167
C03600=1232.557,278.386,-63.937,-176.547,6.500,148.167
C03601=1232.561,278.138,-63.910,-176.549,6.498,148.167
C03602=1232.565,277.889,-63.881,-176.552,6.496,148.168
C03603=1232.570,277.641,-63.854,-176.554,6.494,148.168
C03604=1232.575,277.393,-63.826,-176.557,6.492,148.168
C03605=1232.578,277.144,-63.798,-176.559,6.490,148.168
C03606=1232.583,276.896,-63.770,-176.561,6.488,148.168
C03607=1232.587,276.647,-63.742,-176.564,6.486,148.169
C03608=1232.592,276.399,-63.714,-176.567,6.483,148.169
C03609=1232.596,276.150,-63.686,-176.569,6.481,148.169
C03610=1232.601,275.902,-63.658,-176.571,6.479,148.169
C03611=1232.605,275.654,-63.631,-176.573,6.477,148.169
C03612=1232.609,275.405,-63.603,-176.576,6.475,148.170
C03613=1232.614,275.157,-63.574,-176.578,6.472,148.170
C03614=1232.618,274.908,-63.546,-176.581,6.471,148.170
C03615=1232.623,274.660,-63.519,-176.583,6.468,148.170
C03616=1232.627,274.412,-63.491,-176.585,6.466,148.170
C03617=1232.631,274.163,-63.463,-176.589,6.464,148.170
C03618=1232.636,273.914,-63.435,-176.591,6.461,148.171
C03619=1232.640,273.667,-63.408,-176.593,6.460,148.171
C03620=1232.644,273.418,-63.380,-176.595,6.457,148.171
C03621=1232.649,273.170,-63.352,-176.598,6.455,148.171
C03622=1232.653,272.922,-63.325,-176.600,6.453,148.171
C03623=1232.658,272.672,-63.297,-176.603,6.451,148.172
C03624=1232.662,272.424,-63.269,-176.605,6.449,148.172
C03625=1232.667,272.176,-63.242,-176.607,6.447,148.172
C03626=1232.671,271.927,-63.214,-176.610,6.445,148.172
C03627=1232.675,271.679,-63.186,-176.613,6.442,148.172
C03628=1232.680,271.431,-63.159,-176.615,6.440,148.173
C03629=1232.683,271.182,-63.131,-176.617,6.438,148.173
C03630=1232.689,270.933,-63.103,-176.620,6.436,148.173
C03631=1232.693,270.686,-63.075,-176.623,6.434,148.173
C03632=1232.697,270.436,-63.048,-176.625,6.432,148.173
C03633=1232.702,270.188,-63.020,-176.627,6.430,148.174
C03634=1232.706,269.940,-62.993,-176.629,6.428,148.174
C03635=1232.710,269.691,-62.965,-176.632,6.426,148.174
C03636=1232.715,269.443,-62.938,-176.634,6.424,148.174
C03637=1232.719,269.194,-62.911,-176.637,6.422,148.174
C03638=1232.724,268.947,-62.883,-176.639,6.420,148.175
C03639=1232.728,268.697,-62.856,-176.641,6.418,148.175
C03640=1232.732,268.449,-62.828,-176.645,6.415,148.175
C03641=1232.737,268.201,-62.801,-176.647,6.413,148.175
C03642=1232.741,267.952,-62.774,-176.649,6.411,148.175
C03643=1232.745,267.704,-62.745,-176.652,6.409,148.176
C03644=1232.750,267.455,-62.718,-176.654,6.407,148.176
C03645=1232.754,267.208,-62.691,-176.657,6.405,148.176
C03646=1232.760,266.959,-62.663,-176.659,6.403,148.176
C03647=1232.764,266.710,-62.636,-176.661,6.401,148.176
C03648=1232.767,266.462,-62.608,-176.664,6.399,148.177
C03649=1232.772,266.213,-62.581,-176.667,6.397,148.177
